LIN {X 0,Y 573.567,Z 656.189,A -85,B 0,C 180,E1 -2262.742,E2 -2262.742} C_VEL
LIN {X 0,Y 573.743,Z 644.019,A -85,B 0,C 180,E1 -2263.819,E2 -2263.819} C_VEL
LIN {X 0,Y 573.96,Z 630.902,A -85,B 0,C 180,E1 -2264.781,E2 -2264.781} C_VEL
LIN {X 0,Y 574.111,Z 618.515,A -85,B 0,C 180,E1 -2265.532,E2 -2265.532} C_VEL
LIN {X 0,Y 574.333,Z 603.831,A -85,B 0,C 180,E1 -2266.255,E2 -2266.255} C_VEL
LIN {X 0,Y 574.538,Z 589.615,A -85,B 0,C 180,E1 -2266.798,E2 -2266.798} C_VEL
LIN {X 0,Y 574.7,Z 574.63,A -85,B 0,C 180,E1 -2267.221,E2 -2267.221} C_VEL
LIN {X 0,Y 574.751,Z 559.735,A -85,B 0,C 180,E1 -2267.502,E2 -2267.502} C_VEL
LIN {X 0,Y 575.142,Z 404.764,A -85,B 0,C 180,E1 -2269.493,E2 -2269.493} C_VEL
LIN {X 0,Y 574.007,Z 398.748,A -85,B 0,C 180,E1 -2269.627,E2 -2269.627} C_VEL
LIN {X 0,Y 574.33,Z 374.816,A -85,B 0,C 180,E1 -2272.483,E2 -2272.483} C_VEL
LIN {X 0,Y 574.662,Z 351.3,A -85,B 0,C 180,E1 -2275.343,E2 -2275.343} C_VEL
LIN {X 0,Y 574.14,Z 346.557,A -85,B 0,C 180,E1 -2275.952,E2 -2275.952} C_VEL
LIN {X 0,Y 573.222,Z 342.711,A -85,B 0,C 180,E1 -2276.489,E2 -2276.489} C_VEL
LIN {X 0,Y 573.243,Z 342.7,A -85,B 0,C 180,E1 -2279.367,E2 -2279.367} C_VEL
LIN {X 0,Y 573.248,Z 342.707,A -85,B 0,C 180,E1 -2282.228,E2 -2282.228} C_VEL
LIN {X 0,Y 573.221,Z 342.706,A -85,B 0,C 180,E1 -2284.769,E2 -2284.769} C_VEL
LIN {X 0,Y 573.22,Z 342.704,A -85,B 0,C 180,E1 -2287.809,E2 -2287.809} C_VEL
LIN {X 0,Y 573.245,Z 342.706,A -85,B 0,C 180,E1 -2290.525,E2 -2290.525} C_VEL
LIN {X 0,Y 573.206,Z 342.703,A -85,B 0,C 180,E1 -2293.362,E2 -2293.362} C_VEL
LIN {X 0,Y 573.205,Z 342.713,A -85,B 0,C 180,E1 -2296.335,E2 -2296.335} C_VEL
LIN {X 0,Y 573.205,Z 342.711,A -85,B 0,C 180,E1 -2298.541,E2 -2298.541} C_VEL
LIN {X 0,Y 573.232,Z 342.7,A -85,B 0,C 180,E1 -2301.298,E2 -2301.298} C_VEL
LIN {X 0,Y 573.187,Z 342.708,A -85,B 0,C 180,E1 -2304.022,E2 -2304.022} C_VEL
LIN {X 0,Y 573.254,Z 342.705,A -85,B 0,C 180,E1 -2306.517,E2 -2306.517} C_VEL
LIN {X 0,Y 573.22,Z 342.699,A -85,B 0,C 180,E1 -2309.12,E2 -2309.12} C_VEL
LIN {X 0,Y 573.218,Z 342.705,A -85,B 0,C 180,E1 -2311.978,E2 -2311.978} C_VEL
LIN {X 0,Y 573.235,Z 342.707,A -85,B 0,C 180,E1 -2314.589,E2 -2314.589} C_VEL
LIN {X 0,Y 573.22,Z 342.701,A -85,B 0,C 180,E1 -2317.662,E2 -2317.662} C_VEL
LIN {X 0,Y 573.235,Z 342.702,A -85,B 0,C 180,E1 -2319.923,E2 -2319.923} C_VEL
LIN {X 0,Y 573.239,Z 342.702,A -85,B 0,C 180,E1 -2322.888,E2 -2322.888} C_VEL
LIN {X 0,Y 573.259,Z 342.698,A -85,B 0,C 180,E1 -2325.807,E2 -2325.807} C_VEL
LIN {X 0,Y 573.265,Z 342.701,A -85,B 0,C 180,E1 -2328.745,E2 -2328.745} C_VEL
LIN {X 0,Y 573.25,Z 342.697,A -85,B 0,C 180,E1 -2331.54,E2 -2331.54} C_VEL
LIN {X 0,Y 573.281,Z 342.703,A -85,B 0,C 180,E1 -2334.372,E2 -2334.372} C_VEL
LIN {X 0,Y 573.311,Z 342.692,A -85,B 0,C 180,E1 -2337.893,E2 -2337.893} C_VEL
LIN {X 0,Y 573.327,Z 342.694,A -85,B 0,C 180,E1 -2340.703,E2 -2340.703} C_VEL
LIN {X 0,Y 573.293,Z 342.696,A -85,B 0,C 180,E1 -2342.811,E2 -2342.811} C_VEL
LIN {X 0,Y 573.275,Z 342.695,A -85,B 0,C 180,E1 -2345.629,E2 -2345.629} C_VEL
LIN {X 0,Y 573.254,Z 342.706,A -85,B 0,C 180,E1 -2348.46,E2 -2348.46} C_VEL
LIN {X 0,Y 573.275,Z 342.694,A -85,B 0,C 180,E1 -2351.312,E2 -2351.312} C_VEL
LIN {X 0,Y 573.284,Z 342.703,A -85,B 0,C 180,E1 -2354.424,E2 -2354.424} C_VEL
LIN {X 0,Y 573.258,Z 342.698,A -85,B 0,C 180,E1 -2357.112,E2 -2357.112} C_VEL
LIN {X 0,Y 573.242,Z 342.698,A -85,B 0,C 180,E1 -2360.077,E2 -2360.077} C_VEL
LIN {X 0,Y 573.233,Z 342.707,A -85,B 0,C 180,E1 -2362.338,E2 -2362.338} C_VEL
LIN {X 0,Y 573.228,Z 342.703,A -85,B 0,C 180,E1 -2364.384,E2 -2364.384} C_VEL
LIN {X 0,Y 572.583,Z 342.786,A -85,B 0,C 180,E1 -2364.971,E2 -2364.971} C_VEL
LIN {X 0,Y 569.726,Z 343.142,A -85,B 0,C 180,E1 -2365.922,E2 -2365.922} C_VEL
LIN {X 0,Y 567.296,Z 343.446,A -85,B 0,C 180,E1 -2366.687,E2 -2366.687} C_VEL
LIN {X 0,Y 566.25,Z 343.57,A -85,B 0,C 180,E1 -2367.279,E2 -2367.279} C_VEL
LIN {X 0,Y 566.165,Z 343.58,A -85,B 0,C 180,E1 -2367.479,E2 -2367.479} C_VEL
LIN {X 0,Y 566.202,Z 343.576,A -85,B 0,C 180,E1 -2369.769,E2 -2369.769} C_VEL
LIN {X 0,Y 566.206,Z 343.582,A -85,B 0,C 180,E1 -2372.43,E2 -2372.43} C_VEL
LIN {X 0,Y 566.173,Z 343.58,A -85,B 0,C 180,E1 -2374.988,E2 -2374.988} C_VEL
LIN {X 0,Y 566.19,Z 343.578,A -85,B 0,C 180,E1 -2377.462,E2 -2377.462} C_VEL
LIN {X 0,Y 566.21,Z 343.578,A -85,B 0,C 180,E1 -2380.199,E2 -2380.199} C_VEL
LIN {X 0,Y 566.19,Z 343.58,A -85,B 0,C 180,E1 -2383.056,E2 -2383.056} C_VEL
LIN {X 0,Y 566.197,Z 343.579,A -85,B 0,C 180,E1 -2386.05,E2 -2386.05} C_VEL
LIN {X 0,Y 566.207,Z 343.577,A -85,B 0,C 180,E1 -2389.215,E2 -2389.215} C_VEL
LIN {X 0,Y 566.184,Z 343.579,A -85,B 0,C 180,E1 -2391.637,E2 -2391.637} C_VEL
LIN {X 0,Y 566.153,Z 343.589,A -85,B 0,C 180,E1 -2394.307,E2 -2394.307} C_VEL
LIN {X 0,Y 566.245,Z 343.761,A -85,B 0,C 180,E1 -2396.718,E2 -2396.718} C_VEL
LIN {X 0,Y 567.126,Z 349.166,A -85,B 0,C 180,E1 -2397.534,E2 -2397.534} C_VEL
LIN {X 0,Y 566.884,Z 367.95,A -85,B 0,C 180,E1 -2400.188,E2 -2400.188} C_VEL
LIN {X 0,Y 568.456,Z 375.277,A -85,B 0,C 180,E1 -2400.346,E2 -2400.346} C_VEL
LIN {X 0,Y 567.962,Z 533.328,A -85,B 0,C 180,E1 -2402.415,E2 -2402.415} C_VEL
LIN {X 0,Y 567.836,Z 548.985,A -85,B 0,C 180,E1 -2402.773,E2 -2402.773} C_VEL
LIN {X 0,Y 567.605,Z 564.367,A -85,B 0,C 180,E1 -2403.281,E2 -2403.281} C_VEL
LIN {X 0,Y 567.381,Z 578.806,A -85,B 0,C 180,E1 -2403.913,E2 -2403.913} C_VEL
LIN {X 0,Y 567.142,Z 592.847,A -85,B 0,C 180,E1 -2404.69,E2 -2404.69} C_VEL
LIN {X 0,Y 566.884,Z 605.684,A -85,B 0,C 180,E1 -2405.558,E2 -2405.558} C_VEL
LIN {X 0,Y 566.664,Z 618.585,A -85,B 0,C 180,E1 -2406.617,E2 -2406.617} C_VEL
LIN {X 0,Y 566.45,Z 630.204,A -85,B 0,C 180,E1 -2407.764,E2 -2407.764} C_VEL
LIN {X 0,Y 566.259,Z 639.933,A -85,B 0,C 180,E1 -2408.904,E2 -2408.904} C_VEL
LIN {X 0,Y 566.132,Z 649.359,A -85,B 0,C 180,E1 -2410.228,E2 -2410.228} C_VEL
LIN {X 0,Y 566.048,Z 657.113,A -85,B 0,C 180,E1 -2411.542,E2 -2411.542} C_VEL
LIN {X 0,Y 565.971,Z 663.975,A -85,B 0,C 180,E1 -2412.972,E2 -2412.972} C_VEL
LIN {X 0,Y 565.911,Z 669.753,A -85,B 0,C 180,E1 -2414.514,E2 -2414.514} C_VEL
LIN {X 0,Y 565.895,Z 672.935,A -85,B 0,C 180,E1 -2415.63,E2 -2415.63} C_VEL
LIN {X 0,Y 565.847,Z 676.002,A -85,B 0,C 180,E1 -2417.081,E2 -2417.081} C_VEL
LIN {X 0,Y 565.877,Z 677.854,A -85,B 0,C 180,E1 -2418.538,E2 -2418.538} C_VEL
LIN {X 0,Y 565.88,Z 678.493,A -85,B 0,C 180,E1 -2419.987,E2 -2419.987} C_VEL
LIN {X 0,Y 565.849,Z 677.938,A -85,B 0,C 180,E1 -2421.429,E2 -2421.429} C_VEL
LIN {X 0,Y 565.883,Z 676.229,A -85,B 0,C 180,E1 -2422.866,E2 -2422.866} C_VEL
LIN {X 0,Y 565.921,Z 673.341,A -85,B 0,C 180,E1 -2424.298,E2 -2424.298} C_VEL
LIN {X 0,Y 565.956,Z 669.229,A -85,B 0,C 180,E1 -2425.727,E2 -2425.727} C_VEL
LIN {X 0,Y 565.92,Z 663.819,A -85,B 0,C 180,E1 -2427.153,E2 -2427.153} C_VEL
LIN {X 0,Y 566.009,Z 656.958,A -85,B 0,C 180,E1 -2428.577,E2 -2428.577} C_VEL
LIN {X 0,Y 566.155,Z 648.451,A -85,B 0,C 180,E1 -2430,E2 -2430} C_VEL
LIN {X 0,Y 566.298,Z 639.466,A -85,B 0,C 180,E1 -2431.245,E2 -2431.245} C_VEL
LIN {X 0,Y 566.455,Z 628.688,A -85,B 0,C 180,E1 -2432.489,E2 -2432.489} C_VEL
LIN {X 0,Y 566.681,Z 617.671,A -85,B 0,C 180,E1 -2433.555,E2 -2433.555} C_VEL
LIN {X 0,Y 566.936,Z 605.649,A -85,B 0,C 180,E1 -2434.533,E2 -2434.533} C_VEL
LIN {X 0,Y 567.165,Z 592.496,A -85,B 0,C 180,E1 -2435.422,E2 -2435.422} C_VEL
LIN {X 0,Y 567.403,Z 579.639,A -85,B 0,C 180,E1 -2436.133,E2 -2436.133} C_VEL
LIN {X 0,Y 567.611,Z 565.672,A -85,B 0,C 180,E1 -2436.755,E2 -2436.755} C_VEL
LIN {X 0,Y 567.786,Z 550.58,A -85,B 0,C 180,E1 -2437.27,E2 -2437.27} C_VEL
LIN {X 0,Y 567.906,Z 535.508,A -85,B 0,C 180,E1 -2437.632,E2 -2437.632} C_VEL
LIN {X 0,Y 568.033,Z 511.55,A -85,B 0,C 180,E1 -2437.976,E2 -2437.976} C_VEL
LIN {X 0,Y 568.479,Z 375.352,A -85,B 0,C 180,E1 -2439.742,E2 -2439.742} C_VEL
LIN {X 0,Y 566.9,Z 367.922,A -85,B 0,C 180,E1 -2439.905,E2 -2439.905} C_VEL
LIN {X 0,Y 567.179,Z 349.374,A -85,B 0,C 180,E1 -2442.524,E2 -2442.524} C_VEL
LIN {X 0,Y 566.178,Z 343.589,A -85,B 0,C 180,E1 -2443.413,E2 -2443.413} C_VEL
LIN {X 0,Y 566.185,Z 343.585,A -85,B 0,C 180,E1 -2445.848,E2 -2445.848} C_VEL
LIN {X 0,Y 566.18,Z 343.582,A -85,B 0,C 180,E1 -2448.079,E2 -2448.079} C_VEL
LIN {X 0,Y 566.206,Z 343.575,A -85,B 0,C 180,E1 -2450.338,E2 -2450.338} C_VEL
LIN {X 0,Y 566.171,Z 343.586,A -85,B 0,C 180,E1 -2453.28,E2 -2453.28} C_VEL
LIN {X 0,Y 566.198,Z 343.583,A -85,B 0,C 180,E1 -2455.75,E2 -2455.75} C_VEL
LIN {X 0,Y 566.163,Z 343.582,A -85,B 0,C 180,E1 -2458.193,E2 -2458.193} C_VEL
LIN {X 0,Y 566.189,Z 343.58,A -85,B 0,C 180,E1 -2461.075,E2 -2461.075} C_VEL
LIN {X 0,Y 566.216,Z 343.581,A -85,B 0,C 180,E1 -2463.734,E2 -2463.734} C_VEL
LIN {X 0,Y 566.151,Z 343.581,A -85,B 0,C 180,E1 -2466.574,E2 -2466.574} C_VEL
LIN {X 0,Y 566.212,Z 343.58,A -85,B 0,C 180,E1 -2469.274,E2 -2469.274} C_VEL
LIN {X 0,Y 566.173,Z 343.581,A -85,B 0,C 180,E1 -2472.091,E2 -2472.091} C_VEL
LIN {X 0,Y 566.168,Z 343.582,A -85,B 0,C 180,E1 -2475.037,E2 -2475.037} C_VEL
LIN {X 0,Y 566.183,Z 343.582,A -85,B 0,C 180,E1 -2477.909,E2 -2477.909} C_VEL
LIN {X 0,Y 566.211,Z 343.574,A -85,B 0,C 180,E1 -2480.725,E2 -2480.725} C_VEL
LIN {X 0,Y 566.178,Z 343.586,A -85,B 0,C 180,E1 -2483.428,E2 -2483.428} C_VEL
LIN {X 0,Y 566.201,Z 343.576,A -85,B 0,C 180,E1 -2486.268,E2 -2486.268} C_VEL
LIN {X 0,Y 566.189,Z 343.579,A -85,B 0,C 180,E1 -2488.924,E2 -2488.924} C_VEL
LIN {X 0,Y 566.191,Z 343.578,A -85,B 0,C 180,E1 -2491.856,E2 -2491.856} C_VEL
LIN {X 0,Y 566.188,Z 343.572,A -85,B 0,C 180,E1 -2494.249,E2 -2494.249} C_VEL
LIN {X 0,Y 566.17,Z 343.578,A -85,B 0,C 180,E1 -2496.72,E2 -2496.72} C_VEL
LIN {X 0,Y 566.207,Z 343.584,A -85,B 0,C 180,E1 -2499.662,E2 -2499.662} C_VEL
LIN {X 0,Y 566.183,Z 343.58,A -85,B 0,C 180,E1 -2501.921,E2 -2501.921} C_VEL
LIN {X 0,Y 566.19,Z 343.579,A -85,B 0,C 180,E1 -2504.152,E2 -2504.152} C_VEL
LIN {X 0,Y 566.185,Z 343.578,A -85,B 0,C 180,E1 -2506.358,E2 -2506.358} C_VEL
LIN {X 0,Y 566.236,Z 343.574,A -85,B 0,C 180,E1 -2509.27,E2 -2509.27} C_VEL
LIN {X 0,Y 566.194,Z 343.578,A -85,B 0,C 180,E1 -2512.152,E2 -2512.152} C_VEL
LIN {X 0,Y 566.265,Z 343.567,A -85,B 0,C 180,E1 -2515.016,E2 -2515.016} C_VEL
LIN {X 0,Y 566.282,Z 343.571,A -85,B 0,C 180,E1 -2517.866,E2 -2517.866} C_VEL
LIN {X 0,Y 566.29,Z 343.567,A -85,B 0,C 180,E1 -2520,E2 -2520} C_VEL
LIN {X 0,Y 566.255,Z 343.568,A -85,B 0,C 180,E1 -2522.845,E2 -2522.845} C_VEL
LIN {X 0,Y 566.248,Z 343.578,A -85,B 0,C 180,E1 -2525.698,E2 -2525.698} C_VEL
LIN {X 0,Y 566.2,Z 343.575,A -85,B 0,C 180,E1 -2528.566,E2 -2528.566} C_VEL
LIN {X 0,Y 566.242,Z 343.578,A -85,B 0,C 180,E1 -2531.454,E2 -2531.454} C_VEL
LIN {X 0,Y 566.227,Z 343.572,A -85,B 0,C 180,E1 -2534.502,E2 -2534.502} C_VEL
LIN {X 0,Y 566.162,Z 343.585,A -85,B 0,C 180,E1 -2537.333,E2 -2537.333} C_VEL
LIN {X 0,Y 566.201,Z 343.584,A -85,B 0,C 180,E1 -2539.581,E2 -2539.581} C_VEL
LIN {X 0,Y 566.186,Z 343.582,A -85,B 0,C 180,E1 -2541.863,E2 -2541.863} C_VEL
LIN {X 0,Y 566.183,Z 343.579,A -85,B 0,C 180,E1 -2545.022,E2 -2545.022} C_VEL
LIN {X 0,Y 566.168,Z 343.584,A -85,B 0,C 180,E1 -2547.341,E2 -2547.341} C_VEL
LIN {X 0,Y 566.172,Z 343.587,A -85,B 0,C 180,E1 -2549.77,E2 -2549.77} C_VEL
LIN {X 0,Y 566.2,Z 343.576,A -85,B 0,C 180,E1 -2552.429,E2 -2552.429} C_VEL
LIN {X 0,Y 566.169,Z 343.581,A -85,B 0,C 180,E1 -2554.987,E2 -2554.987} C_VEL
LIN {X 0,Y 566.186,Z 343.585,A -85,B 0,C 180,E1 -2557.461,E2 -2557.461} C_VEL
LIN {X 0,Y 566.206,Z 343.577,A -85,B 0,C 180,E1 -2560.199,E2 -2560.199} C_VEL
LIN {X 0,Y 566.177,Z 343.58,A -85,B 0,C 180,E1 -2563.056,E2 -2563.056} C_VEL
LIN {X 0,Y 566.158,Z 343.585,A -85,B 0,C 180,E1 -2566.053,E2 -2566.053} C_VEL
LIN {X 0,Y 566.158,Z 343.582,A -85,B 0,C 180,E1 -2568.859,E2 -2568.859} C_VEL
LIN {X 0,Y 566.202,Z 343.584,A -85,B 0,C 180,E1 -2571.443,E2 -2571.443} C_VEL
LIN {X 0,Y 566.14,Z 343.585,A -85,B 0,C 180,E1 -2574.306,E2 -2574.306} C_VEL
LIN {X 0,Y 566.203,Z 343.577,A -85,B 0,C 180,E1 -2576.897,E2 -2576.897} C_VEL
LIN {X 0,Y 566.175,Z 343.586,A -85,B 0,C 180,E1 -2579.407,E2 -2579.407} C_VEL
LIN {X 0,Y 566.187,Z 343.587,A -85,B 0,C 180,E1 -2581.856,E2 -2581.856} C_VEL
LIN {X 0,Y 566.174,Z 343.693,A -85,B 0,C 180,E1 -2583.323,E2 -2583.323} C_VEL
LIN {X 0,Y 567.812,Z 351.159,A -85,B 0,C 180,E1 -2584.329,E2 -2584.329} C_VEL
LIN {X 0,Y 567.553,Z 371.68,A -85,B 0,C 180,E1 -2586.849,E2 -2586.849} C_VEL
LIN {X 0,Y 567.151,Z 396.606,A -85,B 0,C 180,E1 -2589.868,E2 -2589.868} C_VEL
LIN {X 0,Y 567.116,Z 398.903,A -85,B 0,C 180,E1 -2590.142,E2 -2590.142} C_VEL
LIN {X 0,Y 568.488,Z 406.26,A -85,B 0,C 180,E1 -2590.289,E2 -2590.289} C_VEL
LIN {X 0,Y 567.984,Z 564.94,A -85,B 0,C 180,E1 -2592.364,E2 -2592.364} C_VEL
LIN {X 0,Y 567.834,Z 580.701,A -85,B 0,C 180,E1 -2592.72,E2 -2592.72} C_VEL
LIN {X 0,Y 567.627,Z 596.036,A -85,B 0,C 180,E1 -2593.223,E2 -2593.223} C_VEL
LIN {X 0,Y 567.461,Z 609.77,A -85,B 0,C 180,E1 -2593.82,E2 -2593.82} C_VEL
LIN {X 0,Y 567.151,Z 623.244,A -85,B 0,C 180,E1 -2594.548,E2 -2594.548} C_VEL
LIN {X 0,Y 566.932,Z 635.518,A -85,B 0,C 180,E1 -2595.359,E2 -2595.359} C_VEL
LIN {X 0,Y 566.672,Z 648.29,A -85,B 0,C 180,E1 -2596.37,E2 -2596.37} C_VEL
LIN {X 0,Y 566.491,Z 659.748,A -85,B 0,C 180,E1 -2597.461,E2 -2597.461} C_VEL
LIN {X 0,Y 566.268,Z 670.311,A -85,B 0,C 180,E1 -2598.659,E2 -2598.659} C_VEL
LIN {X 0,Y 566.209,Z 678.856,A -85,B 0,C 180,E1 -2599.812,E2 -2599.812} C_VEL
LIN {X 0,Y 566.057,Z 686.734,A -85,B 0,C 180,E1 -2601.072,E2 -2601.072} C_VEL
LIN {X 0,Y 565.997,Z 694.089,A -85,B 0,C 180,E1 -2602.508,E2 -2602.508} C_VEL
LIN {X 0,Y 565.958,Z 699.923,A -85,B 0,C 180,E1 -2603.941,E2 -2603.941} C_VEL
LIN {X 0,Y 565.866,Z 703.385,A -85,B 0,C 180,E1 -2605.012,E2 -2605.012} C_VEL
LIN {X 0,Y 565.91,Z 706.89,A -85,B 0,C 180,E1 -2606.44,E2 -2606.44} C_VEL
LIN {X 0,Y 565.839,Z 709.192,A -85,B 0,C 180,E1 -2607.865,E2 -2607.865} C_VEL
LIN {X 0,Y 565.836,Z 710.349,A -85,B 0,C 180,E1 -2609.288,E2 -2609.288} C_VEL
LIN {X 0,Y 565.836,Z 710.349,A -85,B 0,C 180,E1 -2610.712,E2 -2610.712} C_VEL
LIN {X 0,Y 565.838,Z 709.19,A -85,B 0,C 180,E1 -2612.135,E2 -2612.135} C_VEL
LIN {X 0,Y 565.91,Z 706.887,A -85,B 0,C 180,E1 -2613.56,E2 -2613.56} C_VEL
LIN {X 0,Y 565.866,Z 703.386,A -85,B 0,C 180,E1 -2614.988,E2 -2614.988} C_VEL
LIN {X 0,Y 565.942,Z 698.609,A -85,B 0,C 180,E1 -2616.417,E2 -2616.417} C_VEL
LIN {X 0,Y 566.014,Z 692.422,A -85,B 0,C 180,E1 -2617.85,E2 -2617.85} C_VEL
LIN {X 0,Y 566.071,Z 684.647,A -85,B 0,C 180,E1 -2619.288,E2 -2619.288} C_VEL
LIN {X 0,Y 566.239,Z 676.369,A -85,B 0,C 180,E1 -2620.549,E2 -2620.549} C_VEL
LIN {X 0,Y 566.367,Z 666.391,A -85,B 0,C 180,E1 -2621.815,E2 -2621.815} C_VEL
LIN {X 0,Y 566.585,Z 656.188,A -85,B 0,C 180,E1 -2622.901,E2 -2622.901} C_VEL
LIN {X 0,Y 566.8,Z 644.019,A -85,B 0,C 180,E1 -2623.992,E2 -2623.992} C_VEL
LIN {X 0,Y 567.037,Z 631.339,A -85,B 0,C 180,E1 -2624.936,E2 -2624.936} C_VEL
LIN {X 0,Y 567.23,Z 618.513,A -85,B 0,C 180,E1 -2625.726,E2 -2625.726} C_VEL
LIN {X 0,Y 567.515,Z 603.829,A -85,B 0,C 180,E1 -2626.456,E2 -2626.456} C_VEL
LIN {X 0,Y 567.726,Z 589.614,A -85,B 0,C 180,E1 -2627.005,E2 -2627.005} C_VEL
LIN {X 0,Y 567.922,Z 575.27,A -85,B 0,C 180,E1 -2627.417,E2 -2627.417} C_VEL
LIN {X 0,Y 567.983,Z 560.821,A -85,B 0,C 180,E1 -2627.7,E2 -2627.7} C_VEL
LIN {X 0,Y 568.462,Z 405.814,A -85,B 0,C 180,E1 -2629.718,E2 -2629.718} C_VEL
LIN {X 0,Y 567.135,Z 398.804,A -85,B 0,C 180,E1 -2629.868,E2 -2629.868} C_VEL
LIN {X 0,Y 567.494,Z 374.816,A -85,B 0,C 180,E1 -2632.769,E2 -2632.769} C_VEL
LIN {X 0,Y 567.834,Z 352.86,A -85,B 0,C 180,E1 -2635.457,E2 -2635.457} C_VEL
LIN {X 0,Y 567.193,Z 347.931,A -85,B 0,C 180,E1 -2636.096,E2 -2636.096} C_VEL
LIN {X 0,Y 566.168,Z 343.589,A -85,B 0,C 180,E1 -2636.718,E2 -2636.718} C_VEL
LIN {X 0,Y 566.193,Z 343.579,A -85,B 0,C 180,E1 -2639.67,E2 -2639.67} C_VEL
LIN {X 0,Y 566.201,Z 343.586,A -85,B 0,C 180,E1 -2642.43,E2 -2642.43} C_VEL
LIN {X 0,Y 566.165,Z 343.583,A -85,B 0,C 180,E1 -2644.987,E2 -2644.987} C_VEL
LIN {X 0,Y 566.185,Z 343.578,A -85,B 0,C 180,E1 -2647.462,E2 -2647.462} C_VEL
LIN {X 0,Y 566.205,Z 343.582,A -85,B 0,C 180,E1 -2650.199,E2 -2650.199} C_VEL
LIN {X 0,Y 566.186,Z 343.579,A -85,B 0,C 180,E1 -2653.056,E2 -2653.056} C_VEL
LIN {X 0,Y 566.156,Z 343.587,A -85,B 0,C 180,E1 -2656.053,E2 -2656.053} C_VEL
LIN {X 0,Y 566.157,Z 343.585,A -85,B 0,C 180,E1 -2658.859,E2 -2658.859} C_VEL
LIN {X 0,Y 566.202,Z 343.576,A -85,B 0,C 180,E1 -2661.443,E2 -2661.443} C_VEL
LIN {X 0,Y 566.142,Z 343.588,A -85,B 0,C 180,E1 -2664.307,E2 -2664.307} C_VEL
LIN {X 0,Y 566.211,Z 343.577,A -85,B 0,C 180,E1 -2666.897,E2 -2666.897} C_VEL
LIN {X 0,Y 566.169,Z 343.575,A -85,B 0,C 180,E1 -2669.407,E2 -2669.407} C_VEL
LIN {X 0,Y 566.188,Z 343.579,A -85,B 0,C 180,E1 -2671.856,E2 -2671.856} C_VEL
LIN {X 0,Y 566.195,Z 343.583,A -85,B 0,C 180,E1 -2674.25,E2 -2674.25} C_VEL
LIN {X 0,Y 566.166,Z 343.585,A -85,B 0,C 180,E1 -2676.72,E2 -2676.72} C_VEL
LIN {X 0,Y 566.202,Z 343.576,A -85,B 0,C 180,E1 -2679.663,E2 -2679.663} C_VEL
LIN {X 0,Y 566.177,Z 343.581,A -85,B 0,C 180,E1 -2681.921,E2 -2681.921} C_VEL
LIN {X 0,Y 566.188,Z 343.58,A -85,B 0,C 180,E1 -2684.89,E2 -2684.89} C_VEL
LIN {X 0,Y 566.213,Z 343.575,A -85,B 0,C 180,E1 -2687.819,E2 -2687.819} C_VEL
LIN {X 0,Y 566.174,Z 343.582,A -85,B 0,C 180,E1 -2689.992,E2 -2689.992} C_VEL
LIN {X 0,Y 566.212,Z 343.578,A -85,B 0,C 180,E1 -2692.87,E2 -2692.87} C_VEL
LIN {X 0,Y 566.262,Z 343.569,A -85,B 0,C 180,E1 -2695.016,E2 -2695.016} C_VEL
LIN {X 0,Y 566.281,Z 343.568,A -85,B 0,C 180,E1 -2697.867,E2 -2697.867} C_VEL
LIN {X 0,Y 566.297,Z 343.57,A -85,B 0,C 180,E1 -2700.711,E2 -2700.711} C_VEL
LIN {X 0,Y 566.259,Z 343.571,A -85,B 0,C 180,E1 -2702.846,E2 -2702.846} C_VEL
LIN {X 0,Y 566.245,Z 343.571,A -85,B 0,C 180,E1 -2705.699,E2 -2705.699} C_VEL
LIN {X 0,Y 566.204,Z 343.584,A -85,B 0,C 180,E1 -2708.566,E2 -2708.566} C_VEL
LIN {X 0,Y 566.245,Z 343.569,A -85,B 0,C 180,E1 -2711.455,E2 -2711.455} C_VEL
LIN {X 0,Y 566.237,Z 343.58,A -85,B 0,C 180,E1 -2714.506,E2 -2714.506} C_VEL
LIN {X 0,Y 566.196,Z 343.576,A -85,B 0,C 180,E1 -2717.332,E2 -2717.332} C_VEL
LIN {X 0,Y 566.209,Z 343.578,A -85,B 0,C 180,E1 -2720.338,E2 -2720.338} C_VEL
LIN {X 0,Y 566.171,Z 343.58,A -85,B 0,C 180,E1 -2723.281,E2 -2723.281} C_VEL
LIN {X 0,Y 566.192,Z 343.574,A -85,B 0,C 180,E1 -2725.751,E2 -2725.751} C_VEL
LIN {X 0,Y 566.165,Z 343.58,A -85,B 0,C 180,E1 -2727.479,E2 -2727.479} C_VEL
LIN {X 0,Y 565.498,Z 343.668,A -85,B 0,C 180,E1 -2728.073,E2 -2728.073} C_VEL
LIN {X 0,Y 562.649,Z 344.021,A -85,B 0,C 180,E1 -2729.037,E2 -2729.037} C_VEL
LIN {X 0,Y 560.246,Z 344.32,A -85,B 0,C 180,E1 -2729.813,E2 -2729.813} C_VEL
LIN {X 0,Y 559.221,Z 344.452,A -85,B 0,C 180,E1 -2730.412,E2 -2730.412} C_VEL
LIN {X 0,Y 559.14,Z 344.456,A -85,B 0,C 180,E1 -2730.615,E2 -2730.615} C_VEL
LIN {X 0,Y 559.156,Z 344.461,A -85,B 0,C 180,E1 -2732.716,E2 -2732.716} C_VEL
LIN {X 0,Y 559.121,Z 344.455,A -85,B 0,C 180,E1 -2735.325,E2 -2735.325} C_VEL
LIN {X 0,Y 559.129,Z 344.46,A -85,B 0,C 180,E1 -2738.018,E2 -2738.018} C_VEL
LIN {X 0,Y 559.131,Z 344.462,A -85,B 0,C 180,E1 -2740.815,E2 -2740.815} C_VEL
LIN {X 0,Y 559.134,Z 344.458,A -85,B 0,C 180,E1 -2743.195,E2 -2743.195} C_VEL
LIN {X 0,Y 559.139,Z 344.461,A -85,B 0,C 180,E1 -2746.266,E2 -2746.266} C_VEL
LIN {X 0,Y 559.159,Z 344.456,A -85,B 0,C 180,E1 -2749.188,E2 -2749.188} C_VEL
LIN {X 0,Y 559.132,Z 344.46,A -85,B 0,C 180,E1 -2751.982,E2 -2751.982} C_VEL
LIN {X 0,Y 559.131,Z 344.466,A -85,B 0,C 180,E1 -2754.788,E2 -2754.788} C_VEL
LIN {X 0,Y 559.206,Z 344.622,A -85,B 0,C 180,E1 -2756.507,E2 -2756.507} C_VEL
LIN {X 0,Y 560.22,Z 350.036,A -85,B 0,C 180,E1 -2757.355,E2 -2757.355} C_VEL
LIN {X 0,Y 559.978,Z 367.88,A -85,B 0,C 180,E1 -2759.923,E2 -2759.923} C_VEL
LIN {X 0,Y 561.822,Z 377.426,A -85,B 0,C 180,E1 -2760.132,E2 -2760.132} C_VEL
LIN {X 0,Y 561.206,Z 533.216,A -85,B 0,C 180,E1 -2762.194,E2 -2762.194} C_VEL
LIN {X 0,Y 561.059,Z 548.754,A -85,B 0,C 180,E1 -2762.551,E2 -2762.551} C_VEL
LIN {X 0,Y 560.78,Z 563.702,A -85,B 0,C 180,E1 -2763.044,E2 -2763.044} C_VEL
LIN {X 0,Y 560.539,Z 578.009,A -85,B 0,C 180,E1 -2763.671,E2 -2763.671} C_VEL
LIN {X 0,Y 560.252,Z 591.626,A -85,B 0,C 180,E1 -2764.421,E2 -2764.421} C_VEL
LIN {X 0,Y 559.979,Z 605.146,A -85,B 0,C 180,E1 -2765.336,E2 -2765.336} C_VEL
LIN {X 0,Y 559.741,Z 617.059,A -85,B 0,C 180,E1 -2766.31,E2 -2766.31} C_VEL
LIN {X 0,Y 559.452,Z 628.959,A -85,B 0,C 180,E1 -2767.471,E2 -2767.471} C_VEL
LIN {X 0,Y 559.219,Z 638.852,A -85,B 0,C 180,E1 -2768.626,E2 -2768.626} C_VEL
LIN {X 0,Y 559.104,Z 648.484,A -85,B 0,C 180,E1 -2769.969,E2 -2769.969} C_VEL
LIN {X 0,Y 558.975,Z 656.374,A -85,B 0,C 180,E1 -2771.3,E2 -2771.3} C_VEL
LIN {X 0,Y 558.913,Z 661.986,A -85,B 0,C 180,E1 -2772.435,E2 -2772.435} C_VEL
LIN {X 0,Y 558.834,Z 668.026,A -85,B 0,C 180,E1 -2773.938,E2 -2773.938} C_VEL
LIN {X 0,Y 558.806,Z 672.584,A -85,B 0,C 180,E1 -2775.432,E2 -2775.432} C_VEL
LIN {X 0,Y 558.749,Z 675.799,A -85,B 0,C 180,E1 -2776.914,E2 -2776.914} C_VEL
LIN {X 0,Y 558.777,Z 677.745,A -85,B 0,C 180,E1 -2778.391,E2 -2778.391} C_VEL
LIN {X 0,Y 558.777,Z 678.466,A -85,B 0,C 180,E1 -2779.858,E2 -2779.858} C_VEL
LIN {X 0,Y 558.763,Z 678.022,A -85,B 0,C 180,E1 -2781.319,E2 -2781.319} C_VEL
LIN {X 0,Y 558.794,Z 676.425,A -85,B 0,C 180,E1 -2782.775,E2 -2782.775} C_VEL
LIN {X 0,Y 558.829,Z 673.652,A -85,B 0,C 180,E1 -2784.226,E2 -2784.226} C_VEL
LIN {X 0,Y 558.861,Z 669.662,A -85,B 0,C 180,E1 -2785.673,E2 -2785.673} C_VEL
LIN {X 0,Y 558.841,Z 664.36,A -85,B 0,C 180,E1 -2787.117,E2 -2787.117} C_VEL
LIN {X 0,Y 558.927,Z 657.62,A -85,B 0,C 180,E1 -2788.559,E2 -2788.559} C_VEL
LIN {X 0,Y 559.106,Z 649.281,A -85,B 0,C 180,E1 -2790,E2 -2790} C_VEL
LIN {X 0,Y 559.254,Z 640.43,A -85,B 0,C 180,E1 -2791.26,E2 -2791.26} C_VEL
LIN {X 0,Y 559.437,Z 629.869,A -85,B 0,C 180,E1 -2792.52,E2 -2792.52} C_VEL
LIN {X 0,Y 559.69,Z 619.043,A -85,B 0,C 180,E1 -2793.6,E2 -2793.6} C_VEL
LIN {X 0,Y 559.962,Z 607.271,A -85,B 0,C 180,E1 -2794.589,E2 -2794.589} C_VEL
LIN {X 0,Y 560.263,Z 594.444,A -85,B 0,C 180,E1 -2795.489,E2 -2795.489} C_VEL
LIN {X 0,Y 560.471,Z 582.059,A -85,B 0,C 180,E1 -2796.209,E2 -2796.209} C_VEL
LIN {X 0,Y 560.743,Z 567.656,A -85,B 0,C 180,E1 -2796.884,E2 -2796.884} C_VEL
LIN {X 0,Y 560.979,Z 552.45,A -85,B 0,C 180,E1 -2797.428,E2 -2797.428} C_VEL
LIN {X 0,Y 561.135,Z 536.82,A -85,B 0,C 180,E1 -2797.824,E2 -2797.824} C_VEL
LIN {X 0,Y 561.289,Z 516.229,A -85,B 0,C 180,E1 -2798.137,E2 -2798.137} C_VEL
LIN {X 0,Y 561.705,Z 376.067,A -85,B 0,C 180,E1 -2799.98,E2 -2799.98} C_VEL
LIN {X 0,Y 560.012,Z 367.885,A -85,B 0,C 180,E1 -2800.165,E2 -2800.165} C_VEL
LIN {X 0,Y 560.244,Z 350.387,A -85,B 0,C 180,E1 -2802.681,E2 -2802.681} C_VEL
LIN {X 0,Y 559.165,Z 344.463,A -85,B 0,C 180,E1 -2803.631,E2 -2803.631} C_VEL
LIN {X 0,Y 559.143,Z 344.46,A -85,B 0,C 180,E1 -2806.053,E2 -2806.053} C_VEL
LIN {X 0,Y 559.162,Z 344.458,A -85,B 0,C 180,E1 -2809.074,E2 -2809.074} C_VEL
LIN {X 0,Y 559.159,Z 344.462,A -85,B 0,C 180,E1 -2811.549,E2 -2811.549} C_VEL
LIN {X 0,Y 559.129,Z 344.457,A -85,B 0,C 180,E1 -2814.507,E2 -2814.507} C_VEL
LIN {X 0,Y 559.137,Z 344.457,A -85,B 0,C 180,E1 -2816.904,E2 -2816.904} C_VEL
LIN {X 0,Y 559.126,Z 344.462,A -85,B 0,C 180,E1 -2819.852,E2 -2819.852} C_VEL
LIN {X 0,Y 559.158,Z 344.452,A -85,B 0,C 180,E1 -2822.715,E2 -2822.715} C_VEL
LIN {X 0,Y 559.122,Z 344.464,A -85,B 0,C 180,E1 -2825.325,E2 -2825.325} C_VEL
LIN {X 0,Y 559.129,Z 344.46,A -85,B 0,C 180,E1 -2828.018,E2 -2828.018} C_VEL
LIN {X 0,Y 559.162,Z 344.454,A -85,B 0,C 180,E1 -2829.941,E2 -2829.941} C_VEL
LIN {X 0,Y 559.144,Z 344.455,A -85,B 0,C 180,E1 -2832.745,E2 -2832.745} C_VEL
LIN {X 0,Y 559.127,Z 344.461,A -85,B 0,C 180,E1 -2835.764,E2 -2835.764} C_VEL
LIN {X 0,Y 559.129,Z 344.458,A -85,B 0,C 180,E1 -2838.226,E2 -2838.226} C_VEL
LIN {X 0,Y 559.173,Z 344.455,A -85,B 0,C 180,E1 -2841.192,E2 -2841.192} C_VEL
LIN {X 0,Y 559.12,Z 344.464,A -85,B 0,C 180,E1 -2843.787,E2 -2843.787} C_VEL
LIN {X 0,Y 559.152,Z 344.453,A -85,B 0,C 180,E1 -2846.424,E2 -2846.424} C_VEL
LIN {X 0,Y 559.154,Z 344.456,A -85,B 0,C 180,E1 -2848.98,E2 -2848.98} C_VEL
LIN {X 0,Y 559.137,Z 344.46,A -85,B 0,C 180,E1 -2851.625,E2 -2851.625} C_VEL
LIN {X 0,Y 559.142,Z 344.449,A -85,B 0,C 180,E1 -2854.822,E2 -2854.822} C_VEL
LIN {X 0,Y 559.142,Z 344.461,A -85,B 0,C 180,E1 -2857.847,E2 -2857.847} C_VEL
LIN {X 0,Y 559.196,Z 344.448,A -85,B 0,C 180,E1 -2860.494,E2 -2860.494} C_VEL
LIN {X 0,Y 559.17,Z 344.453,A -85,B 0,C 180,E1 -2863.197,E2 -2863.197} C_VEL
LIN {X 0,Y 559.161,Z 344.454,A -85,B 0,C 180,E1 -2866.183,E2 -2866.183} C_VEL
LIN {X 0,Y 559.194,Z 344.448,A -85,B 0,C 180,E1 -2869.133,E2 -2869.133} C_VEL
LIN {X 0,Y 559.147,Z 344.457,A -85,B 0,C 180,E1 -2872.052,E2 -2872.052} C_VEL
LIN {X 0,Y 559.24,Z 344.442,A -85,B 0,C 180,E1 -2874.953,E2 -2874.953} C_VEL
LIN {X 0,Y 559.253,Z 344.447,A -85,B 0,C 180,E1 -2877.839,E2 -2877.839} C_VEL
LIN {X 0,Y 559.259,Z 344.443,A -85,B 0,C 180,E1 -2880,E2 -2880} C_VEL
LIN {X 0,Y 559.223,Z 344.444,A -85,B 0,C 180,E1 -2882.881,E2 -2882.881} C_VEL
LIN {X 0,Y 559.217,Z 344.452,A -85,B 0,C 180,E1 -2885.77,E2 -2885.77} C_VEL
LIN {X 0,Y 559.164,Z 344.451,A -85,B 0,C 180,E1 -2888.674,E2 -2888.674} C_VEL
LIN {X 0,Y 559.203,Z 344.456,A -85,B 0,C 180,E1 -2891.6,E2 -2891.6} C_VEL
LIN {X 0,Y 559.183,Z 344.449,A -85,B 0,C 180,E1 -2894.587,E2 -2894.587} C_VEL
LIN {X 0,Y 559.117,Z 344.466,A -85,B 0,C 180,E1 -2897.558,E2 -2897.558} C_VEL
LIN {X 0,Y 559.164,Z 344.458,A -85,B 0,C 180,E1 -2899.837,E2 -2899.837} C_VEL
LIN {X 0,Y 559.132,Z 344.457,A -85,B 0,C 180,E1 -2902.153,E2 -2902.153} C_VEL
LIN {X 0,Y 559.142,Z 344.458,A -85,B 0,C 180,E1 -2905.178,E2 -2905.178} C_VEL
LIN {X 0,Y 559.118,Z 344.467,A -85,B 0,C 180,E1 -2907.715,E2 -2907.715} C_VEL
LIN {X 0,Y 559.137,Z 344.458,A -85,B 0,C 180,E1 -2910.183,E2 -2910.183} C_VEL
LIN {X 0,Y 559.154,Z 344.453,A -85,B 0,C 180,E1 -2912.715,E2 -2912.715} C_VEL
LIN {X 0,Y 559.118,Z 344.463,A -85,B 0,C 180,E1 -2915.325,E2 -2915.325} C_VEL
LIN {X 0,Y 559.124,Z 344.46,A -85,B 0,C 180,E1 -2918.018,E2 -2918.018} C_VEL
LIN {X 0,Y 559.159,Z 344.458,A -85,B 0,C 180,E1 -2919.941,E2 -2919.941} C_VEL
LIN {X 0,Y 559.139,Z 344.455,A -85,B 0,C 180,E1 -2922.745,E2 -2922.745} C_VEL
LIN {X 0,Y 559.124,Z 344.466,A -85,B 0,C 180,E1 -2925.764,E2 -2925.764} C_VEL
LIN {X 0,Y 559.126,Z 344.46,A -85,B 0,C 180,E1 -2928.226,E2 -2928.226} C_VEL
LIN {X 0,Y 559.169,Z 344.456,A -85,B 0,C 180,E1 -2931.192,E2 -2931.192} C_VEL
LIN {X 0,Y 559.115,Z 344.467,A -85,B 0,C 180,E1 -2933.787,E2 -2933.787} C_VEL
LIN {X 0,Y 559.147,Z 344.456,A -85,B 0,C 180,E1 -2936.424,E2 -2936.424} C_VEL
LIN {X 0,Y 559.152,Z 344.456,A -85,B 0,C 180,E1 -2938.98,E2 -2938.98} C_VEL
LIN {X 0,Y 559.133,Z 344.466,A -85,B 0,C 180,E1 -2941.625,E2 -2941.625} C_VEL
LIN {X 0,Y 559.144,Z 344.576,A -85,B 0,C 180,E1 -2943.096,E2 -2943.096} C_VEL
LIN {X 0,Y 560.986,Z 353.201,A -85,B 0,C 180,E1 -2944.272,E2 -2944.272} C_VEL
LIN {X 0,Y 560.69,Z 373.186,A -85,B 0,C 180,E1 -2946.744,E2 -2946.744} C_VEL
LIN {X 0,Y 560.26,Z 397.26,A -85,B 0,C 180,E1 -2949.689,E2 -2949.689} C_VEL
LIN {X 0,Y 560.268,Z 399.043,A -85,B 0,C 180,E1 -2949.891,E2 -2949.891} C_VEL
LIN {X 0,Y 561.819,Z 407.764,A -85,B 0,C 180,E1 -2950.065,E2 -2950.065} C_VEL
LIN {X 0,Y 561.232,Z 565.013,A -85,B 0,C 180,E1 -2952.146,E2 -2952.146} C_VEL
LIN {X 0,Y 561.073,Z 580.224,A -85,B 0,C 180,E1 -2952.492,E2 -2952.492} C_VEL
LIN {X 0,Y 560.832,Z 594.795,A -85,B 0,C 180,E1 -2952.967,E2 -2952.967} C_VEL
LIN {X 0,Y 560.659,Z 607.801,A -85,B 0,C 180,E1 -2953.524,E2 -2953.524} C_VEL
LIN {X 0,Y 560.317,Z 621.676,A -85,B 0,C 180,E1 -2954.262,E2 -2954.262} C_VEL
LIN {X 0,Y 560.021,Z 635.519,A -85,B 0,C 180,E1 -2955.174,E2 -2955.174} C_VEL
LIN {X 0,Y 559.722,Z 648.291,A -85,B 0,C 180,E1 -2956.198,E2 -2956.198} C_VEL
LIN {X 0,Y 559.516,Z 659.748,A -85,B 0,C 180,E1 -2957.302,E2 -2957.302} C_VEL
LIN {X 0,Y 559.304,Z 669.389,A -85,B 0,C 180,E1 -2958.402,E2 -2958.402} C_VEL
LIN {X 0,Y 559.168,Z 678.855,A -85,B 0,C 180,E1 -2959.682,E2 -2959.682} C_VEL
LIN {X 0,Y 559.002,Z 686.734,A -85,B 0,C 180,E1 -2960.958,E2 -2960.958} C_VEL
LIN {X 0,Y 558.92,Z 694.089,A -85,B 0,C 180,E1 -2962.413,E2 -2962.413} C_VEL
LIN {X 0,Y 558.859,Z 699.922,A -85,B 0,C 180,E1 -2963.864,E2 -2963.864} C_VEL
LIN {X 0,Y 558.787,Z 703.386,A -85,B 0,C 180,E1 -2964.949,E2 -2964.949} C_VEL
LIN {X 0,Y 558.819,Z 706.889,A -85,B 0,C 180,E1 -2966.395,E2 -2966.395} C_VEL
LIN {X 0,Y 558.744,Z 709.191,A -85,B 0,C 180,E1 -2967.837,E2 -2967.837} C_VEL
LIN {X 0,Y 558.737,Z 710.349,A -85,B 0,C 180,E1 -2969.279,E2 -2969.279} C_VEL
LIN {X 0,Y 558.737,Z 710.348,A -85,B 0,C 180,E1 -2970.721,E2 -2970.721} C_VEL
LIN {X 0,Y 558.744,Z 709.189,A -85,B 0,C 180,E1 -2972.163,E2 -2972.163} C_VEL
LIN {X 0,Y 558.819,Z 706.886,A -85,B 0,C 180,E1 -2973.605,E2 -2973.605} C_VEL
LIN {X 0,Y 558.787,Z 703.386,A -85,B 0,C 180,E1 -2975.051,E2 -2975.051} C_VEL
LIN {X 0,Y 558.85,Z 698.609,A -85,B 0,C 180,E1 -2976.499,E2 -2976.499} C_VEL
LIN {X 0,Y 558.95,Z 692.422,A -85,B 0,C 180,E1 -2977.95,E2 -2977.95} C_VEL
LIN {X 0,Y 559.005,Z 684.646,A -85,B 0,C 180,E1 -2979.407,E2 -2979.407} C_VEL
LIN {X 0,Y 559.217,Z 676.368,A -85,B 0,C 180,E1 -2980.683,E2 -2980.683} C_VEL
LIN {X 0,Y 559.362,Z 666.391,A -85,B 0,C 180,E1 -2981.965,E2 -2981.965} C_VEL
LIN {X 0,Y 559.596,Z 656.187,A -85,B 0,C 180,E1 -2983.065,E2 -2983.065} C_VEL
LIN {X 0,Y 559.862,Z 644.019,A -85,B 0,C 180,E1 -2984.169,E2 -2984.169} C_VEL
LIN {X 0,Y 560.123,Z 631.688,A -85,B 0,C 180,E1 -2985.1,E2 -2985.1} C_VEL
LIN {X 0,Y 560.359,Z 618.51,A -85,B 0,C 180,E1 -2985.924,E2 -2985.924} C_VEL
LIN {X 0,Y 560.677,Z 603.826,A -85,B 0,C 180,E1 -2986.663,E2 -2986.663} C_VEL
LIN {X 0,Y 560.916,Z 589.614,A -85,B 0,C 180,E1 -2987.218,E2 -2987.218} C_VEL
LIN {X 0,Y 561.142,Z 575.248,A -85,B 0,C 180,E1 -2987.635,E2 -2987.635} C_VEL
LIN {X 0,Y 561.227,Z 560.813,A -85,B 0,C 180,E1 -2987.921,E2 -2987.921} C_VEL
LIN {X 0,Y 561.782,Z 406.846,A -85,B 0,C 180,E1 -2989.949,E2 -2989.949} C_VEL
LIN {X 0,Y 560.241,Z 398.88,A -85,B 0,C 180,E1 -2990.113,E2 -2990.113} C_VEL
LIN {X 0,Y 560.648,Z 374.764,A -85,B 0,C 180,E1 -2993.062,E2 -2993.062} C_VEL
LIN {X 0,Y 561.004,Z 354.32,A -85,B 0,C 180,E1 -2995.58,E2 -2995.58} C_VEL
LIN {X 0,Y 560.66,Z 350.91,A -85,B 0,C 180,E1 -2996.023,E2 -2996.023} C_VEL
LIN {X 0,Y 559.121,Z 344.466,A -85,B 0,C 180,E1 -2996.93,E2 -2996.93} C_VEL
LIN {X 0,Y 559.14,Z 344.46,A -85,B 0,C 180,E1 -2999.856,E2 -2999.856} C_VEL
LIN {X 0,Y 559.152,Z 344.46,A -85,B 0,C 180,E1 -3002.716,E2 -3002.716} C_VEL
LIN {X 0,Y 559.115,Z 344.46,A -85,B 0,C 180,E1 -3005.325,E2 -3005.325} C_VEL
LIN {X 0,Y 559.124,Z 344.463,A -85,B 0,C 180,E1 -3008.018,E2 -3008.018} C_VEL
LIN {X 0,Y 559.126,Z 344.46,A -85,B 0,C 180,E1 -3010.815,E2 -3010.815} C_VEL
LIN {X 0,Y 559.129,Z 344.458,A -85,B 0,C 180,E1 -3013.195,E2 -3013.195} C_VEL
LIN {X 0,Y 559.123,Z 344.46,A -85,B 0,C 180,E1 -3015.764,E2 -3015.764} C_VEL
LIN {X 0,Y 559.12,Z 344.466,A -85,B 0,C 180,E1 -3018.226,E2 -3018.226} C_VEL
LIN {X 0,Y 559.169,Z 344.452,A -85,B 0,C 180,E1 -3021.193,E2 -3021.193} C_VEL
LIN {X 0,Y 559.116,Z 344.457,A -85,B 0,C 180,E1 -3023.788,E2 -3023.788} C_VEL
LIN {X 0,Y 559.16,Z 344.462,A -85,B 0,C 180,E1 -3026.425,E2 -3026.425} C_VEL
LIN {X 0,Y 559.149,Z 344.451,A -85,B 0,C 180,E1 -3028.981,E2 -3028.981} C_VEL
LIN {X 0,Y 559.133,Z 344.456,A -85,B 0,C 180,E1 -3031.626,E2 -3031.626} C_VEL
LIN {X 0,Y 559.16,Z 344.455,A -85,B 0,C 180,E1 -3033.902,E2 -3033.902} C_VEL
LIN {X 0,Y 559.135,Z 344.463,A -85,B 0,C 180,E1 -3036.573,E2 -3036.573} C_VEL
LIN {X 0,Y 559.173,Z 344.451,A -85,B 0,C 180,E1 -3039.395,E2 -3039.395} C_VEL
LIN {X 0,Y 559.125,Z 344.458,A -85,B 0,C 180,E1 -3041.685,E2 -3041.685} C_VEL
LIN {X 0,Y 559.139,Z 344.458,A -85,B 0,C 180,E1 -3043.947,E2 -3043.947} C_VEL
LIN {X 0,Y 559.157,Z 344.459,A -85,B 0,C 180,E1 -3046.184,E2 -3046.184} C_VEL
LIN {X 0,Y 559.192,Z 344.45,A -85,B 0,C 180,E1 -3049.134,E2 -3049.134} C_VEL
LIN {X 0,Y 559.191,Z 344.452,A -85,B 0,C 180,E1 -3052.054,E2 -3052.054} C_VEL
LIN {X 0,Y 559.238,Z 344.444,A -85,B 0,C 180,E1 -3054.953,E2 -3054.953} C_VEL
LIN {X 0,Y 559.252,Z 344.443,A -85,B 0,C 180,E1 -3057.84,E2 -3057.84} C_VEL
LIN {X 0,Y 559.268,Z 344.445,A -85,B 0,C 180,E1 -3060.72,E2 -3060.72} C_VEL
LIN {X 0,Y 559.225,Z 344.447,A -85,B 0,C 180,E1 -3062.882,E2 -3062.882} C_VEL
LIN {X 0,Y 559.215,Z 344.447,A -85,B 0,C 180,E1 -3065.771,E2 -3065.771} C_VEL
LIN {X 0,Y 559.168,Z 344.459,A -85,B 0,C 180,E1 -3068.675,E2 -3068.675} C_VEL
LIN {X 0,Y 559.207,Z 344.446,A -85,B 0,C 180,E1 -3071.601,E2 -3071.601} C_VEL
LIN {X 0,Y 559.204,Z 344.456,A -85,B 0,C 180,E1 -3074.596,E2 -3074.596} C_VEL
LIN {X 0,Y 559.14,Z 344.455,A -85,B 0,C 180,E1 -3077.558,E2 -3077.558} C_VEL
LIN {X 0,Y 559.168,Z 344.448,A -85,B 0,C 180,E1 -3079.838,E2 -3079.838} C_VEL
LIN {X 0,Y 559.142,Z 344.459,A -85,B 0,C 180,E1 -3082.153,E2 -3082.153} C_VEL
LIN {X 0,Y 559.144,Z 344.452,A -85,B 0,C 180,E1 -3085.179,E2 -3085.179} C_VEL
LIN {X 0,Y 559.137,Z 344.463,A -85,B 0,C 180,E1 -3088.375,E2 -3088.375} C_VEL
LIN {X 0,Y 559.14,Z 344.456,A -85,B 0,C 180,E1 -3090.615,E2 -3090.615} C_VEL
LIN {X 0,Y 558.479,Z 344.538,A -85,B 0,C 180,E1 -3091.216,E2 -3091.216} C_VEL
LIN {X 0,Y 555.615,Z 344.897,A -85,B 0,C 180,E1 -3092.192,E2 -3092.192} C_VEL
LIN {X 0,Y 553.198,Z 345.199,A -85,B 0,C 180,E1 -3092.978,E2 -3092.978} C_VEL
LIN {X 0,Y 552.171,Z 345.325,A -85,B 0,C 180,E1 -3093.584,E2 -3093.584} C_VEL
LIN {X 0,Y 552.093,Z 345.335,A -85,B 0,C 180,E1 -3093.79,E2 -3093.79} C_VEL
LIN {X 0,Y 552.1,Z 345.34,A -85,B 0,C 180,E1 -3096.748,E2 -3096.748} C_VEL
LIN {X 0,Y 552.13,Z 345.327,A -85,B 0,C 180,E1 -3099.528,E2 -3099.528} C_VEL
LIN {X 0,Y 552.112,Z 345.338,A -85,B 0,C 180,E1 -3102.428,E2 -3102.428} C_VEL
LIN {X 0,Y 552.095,Z 345.333,A -85,B 0,C 180,E1 -3105.562,E2 -3105.562} C_VEL
LIN {X 0,Y 552.112,Z 345.34,A -85,B 0,C 180,E1 -3108.68,E2 -3108.68} C_VEL
LIN {X 0,Y 552.118,Z 345.332,A -85,B 0,C 180,E1 -3111.411,E2 -3111.411} C_VEL
LIN {X 0,Y 552.078,Z 345.341,A -85,B 0,C 180,E1 -3114.156,E2 -3114.156} C_VEL
LIN {X 0,Y 552.142,Z 345.353,A -85,B 0,C 180,E1 -3116.27,E2 -3116.27} C_VEL
LIN {X 0,Y 553.364,Z 352.057,A -85,B 0,C 180,E1 -3117.332,E2 -3117.332} C_VEL
LIN {X 0,Y 553.054,Z 368.068,A -85,B 0,C 180,E1 -3119.675,E2 -3119.675} C_VEL
LIN {X 0,Y 555.15,Z 377.729,A -85,B 0,C 180,E1 -3119.887,E2 -3119.887} C_VEL
LIN {X 0,Y 554.435,Z 533.074,A -85,B 0,C 180,E1 -3121.966,E2 -3121.966} C_VEL
LIN {X 0,Y 554.266,Z 549.008,A -85,B 0,C 180,E1 -3122.337,E2 -3122.337} C_VEL
LIN {X 0,Y 553.989,Z 563.616,A -85,B 0,C 180,E1 -3122.825,E2 -3122.825} C_VEL
LIN {X 0,Y 553.696,Z 577.16,A -85,B 0,C 180,E1 -3123.421,E2 -3123.421} C_VEL
LIN {X 0,Y 553.388,Z 591.871,A -85,B 0,C 180,E1 -3124.237,E2 -3124.237} C_VEL
LIN {X 0,Y 553.054,Z 604.592,A -85,B 0,C 180,E1 -3125.106,E2 -3125.106} C_VEL
LIN {X 0,Y 552.774,Z 617.595,A -85,B 0,C 180,E1 -3126.181,E2 -3126.181} C_VEL
LIN {X 0,Y 552.442,Z 629.493,A -85,B 0,C 180,E1 -3127.367,E2 -3127.367} C_VEL
LIN {X 0,Y 552.208,Z 639.314,A -85,B 0,C 180,E1 -3128.537,E2 -3128.537} C_VEL
LIN {X 0,Y 552.068,Z 648.865,A -85,B 0,C 180,E1 -3129.896,E2 -3129.896} C_VEL
LIN {X 0,Y 551.898,Z 656.684,A -85,B 0,C 180,E1 -3131.244,E2 -3131.244} C_VEL
LIN {X 0,Y 551.815,Z 663.969,A -85,B 0,C 180,E1 -3132.789,E2 -3132.789} C_VEL
LIN {X 0,Y 551.753,Z 668.86,A -85,B 0,C 180,E1 -3134.106,E2 -3134.106} C_VEL
LIN {X 0,Y 551.713,Z 672.889,A -85,B 0,C 180,E1 -3135.497,E2 -3135.497} C_VEL
LIN {X 0,Y 551.664,Z 675.575,A -85,B 0,C 180,E1 -3136.743,E2 -3136.743} C_VEL
LIN {X 0,Y 551.674,Z 677.606,A -85,B 0,C 180,E1 -3138.239,E2 -3138.239} C_VEL
LIN {X 0,Y 551.674,Z 678.438,A -85,B 0,C 180,E1 -3139.726,E2 -3139.726} C_VEL
LIN {X 0,Y 551.668,Z 678.106,A -85,B 0,C 180,E1 -3141.206,E2 -3141.206} C_VEL
LIN {X 0,Y 551.69,Z 676.62,A -85,B 0,C 180,E1 -3142.681,E2 -3142.681} C_VEL
LIN {X 0,Y 551.744,Z 673.963,A -85,B 0,C 180,E1 -3144.151,E2 -3144.151} C_VEL
LIN {X 0,Y 551.75,Z 670.06,A -85,B 0,C 180,E1 -3145.617,E2 -3145.617} C_VEL
LIN {X 0,Y 551.765,Z 664.856,A -85,B 0,C 180,E1 -3147.08,E2 -3147.08} C_VEL
LIN {X 0,Y 551.842,Z 658.254,A -85,B 0,C 180,E1 -3148.54,E2 -3148.54} C_VEL
LIN {X 0,Y 552.006,Z 651.167,A -85,B 0,C 180,E1 -3149.818,E2 -3149.818} C_VEL
LIN {X 0,Y 552.163,Z 642.707,A -85,B 0,C 180,E1 -3151.094,E2 -3151.094} C_VEL
LIN {X 0,Y 552.4,Z 632.586,A -85,B 0,C 180,E1 -3152.37,E2 -3152.37} C_VEL
LIN {X 0,Y 552.651,Z 622.297,A -85,B 0,C 180,E1 -3153.463,E2 -3153.463} C_VEL
LIN {X 0,Y 552.968,Z 610.027,A -85,B 0,C 180,E1 -3154.556,E2 -3154.556} C_VEL
LIN {X 0,Y 553.31,Z 597.778,A -85,B 0,C 180,E1 -3155.467,E2 -3155.467} C_VEL
LIN {X 0,Y 553.593,Z 584.456,A -85,B 0,C 180,E1 -3156.286,E2 -3156.286} C_VEL
LIN {X 0,Y 553.888,Z 569.634,A -85,B 0,C 180,E1 -3157.015,E2 -3157.015} C_VEL
LIN {X 0,Y 554.154,Z 554.526,A -85,B 0,C 180,E1 -3157.584,E2 -3157.584} C_VEL
LIN {X 0,Y 554.428,Z 539.419,A -85,B 0,C 180,E1 -3157.992,E2 -3157.992} C_VEL
LIN {X 0,Y 554.524,Z 524.9,A -85,B 0,C 180,E1 -3158.25,E2 -3158.25} C_VEL
LIN {X 0,Y 555.081,Z 377.431,A -85,B 0,C 180,E1 -3160.21,E2 -3160.21} C_VEL
LIN {X 0,Y 553.096,Z 367.898,A -85,B 0,C 180,E1 -3160.432,E2 -3160.432} C_VEL
LIN {X 0,Y 553.419,Z 352.72,A -85,B 0,C 180,E1 -3162.654,E2 -3162.654} C_VEL
LIN {X 0,Y 552.121,Z 345.339,A -85,B 0,C 180,E1 -3163.855,E2 -3163.855} C_VEL
LIN {X 0,Y 552.113,Z 345.336,A -85,B 0,C 180,E1 -3167.024,E2 -3167.024} C_VEL
LIN {X 0,Y 552.13,Z 345.331,A -85,B 0,C 180,E1 -3170.101,E2 -3170.101} C_VEL
LIN {X 0,Y 552.089,Z 345.335,A -85,B 0,C 180,E1 -3172.451,E2 -3172.451} C_VEL
LIN {X 0,Y 552.09,Z 345.341,A -85,B 0,C 180,E1 -3175.334,E2 -3175.334} C_VEL
LIN {X 0,Y 552.068,Z 345.339,A -85,B 0,C 180,E1 -3178.101,E2 -3178.101} C_VEL
LIN {X 0,Y 552.097,Z 345.333,A -85,B 0,C 180,E1 -3180.61,E2 -3180.61} C_VEL
LIN {X 0,Y 552.118,Z 345.333,A -85,B 0,C 180,E1 -3183.186,E2 -3183.186} C_VEL
LIN {X 0,Y 552.074,Z 345.339,A -85,B 0,C 180,E1 -3185.845,E2 -3185.845} C_VEL
LIN {X 0,Y 552.122,Z 345.333,A -85,B 0,C 180,E1 -3189.06,E2 -3189.06} C_VEL
LIN {X 0,Y 552.08,Z 345.34,A -85,B 0,C 180,E1 -3191.45,E2 -3191.45} C_VEL
LIN {X 0,Y 552.079,Z 345.334,A -85,B 0,C 180,E1 -3194.529,E2 -3194.529} C_VEL
LIN {X 0,Y 552.113,Z 345.339,A -85,B 0,C 180,E1 -3197.587,E2 -3197.587} C_VEL
LIN {X 0,Y 552.13,Z 345.328,A -85,B 0,C 180,E1 -3200.472,E2 -3200.472} C_VEL
LIN {X 0,Y 552.1,Z 345.338,A -85,B 0,C 180,E1 -3203.318,E2 -3203.318} C_VEL
LIN {X 0,Y 552.104,Z 345.335,A -85,B 0,C 180,E1 -3205.937,E2 -3205.937} C_VEL
LIN {X 0,Y 552.124,Z 345.33,A -85,B 0,C 180,E1 -3208.54,E2 -3208.54} C_VEL
LIN {X 0,Y 552.099,Z 345.339,A -85,B 0,C 180,E1 -3211.443,E2 -3211.443} C_VEL
LIN {X 0,Y 552.081,Z 345.327,A -85,B 0,C 180,E1 -3214.353,E2 -3214.353} C_VEL
LIN {X 0,Y 552.097,Z 345.33,A -85,B 0,C 180,E1 -3216.757,E2 -3216.757} C_VEL
LIN {X 0,Y 552.121,Z 345.333,A -85,B 0,C 180,E1 -3219.119,E2 -3219.119} C_VEL
LIN {X 0,Y 552.091,Z 345.341,A -85,B 0,C 180,E1 -3221.443,E2 -3221.443} C_VEL
LIN {X 0,Y 552.105,Z 345.339,A -85,B 0,C 180,E1 -3223.737,E2 -3223.737} C_VEL
LIN {X 0,Y 552.129,Z 345.332,A -85,B 0,C 180,E1 -3226.004,E2 -3226.004} C_VEL
LIN {X 0,Y 552.163,Z 345.323,A -85,B 0,C 180,E1 -3228.993,E2 -3228.993} C_VEL
LIN {X 0,Y 552.116,Z 345.334,A -85,B 0,C 180,E1 -3231.951,E2 -3231.951} C_VEL
LIN {X 0,Y 552.216,Z 345.316,A -85,B 0,C 180,E1 -3234.888,E2 -3234.888} C_VEL
LIN {X 0,Y 552.224,Z 345.323,A -85,B 0,C 180,E1 -3237.812,E2 -3237.812} C_VEL
LIN {X 0,Y 552.228,Z 345.318,A -85,B 0,C 180,E1 -3240,E2 -3240} C_VEL
LIN {X 0,Y 552.191,Z 345.32,A -85,B 0,C 180,E1 -3242.918,E2 -3242.918} C_VEL
LIN {X 0,Y 552.187,Z 345.327,A -85,B 0,C 180,E1 -3245.844,E2 -3245.844} C_VEL
LIN {X 0,Y 552.136,Z 345.327,A -85,B 0,C 180,E1 -3248.786,E2 -3248.786} C_VEL
LIN {X 0,Y 552.159,Z 345.331,A -85,B 0,C 180,E1 -3251.75,E2 -3251.75} C_VEL
LIN {X 0,Y 552.13,Z 345.328,A -85,B 0,C 180,E1 -3254.748,E2 -3254.748} C_VEL
LIN {X 0,Y 552.081,Z 345.34,A -85,B 0,C 180,E1 -3257.789,E2 -3257.789} C_VEL
LIN {X 0,Y 552.125,Z 345.331,A -85,B 0,C 180,E1 -3260.101,E2 -3260.101} C_VEL
LIN {X 0,Y 552.084,Z 345.333,A -85,B 0,C 180,E1 -3262.451,E2 -3262.451} C_VEL
LIN {X 0,Y 552.086,Z 345.339,A -85,B 0,C 180,E1 -3265.334,E2 -3265.334} C_VEL
LIN {X 0,Y 552.064,Z 345.34,A -85,B 0,C 180,E1 -3268.101,E2 -3268.101} C_VEL
LIN {X 0,Y 552.093,Z 345.333,A -85,B 0,C 180,E1 -3270.61,E2 -3270.61} C_VEL
LIN {X 0,Y 552.114,Z 345.333,A -85,B 0,C 180,E1 -3273.186,E2 -3273.186} C_VEL
LIN {X 0,Y 552.07,Z 345.343,A -85,B 0,C 180,E1 -3275.845,E2 -3275.845} C_VEL
LIN {X 0,Y 552.117,Z 345.331,A -85,B 0,C 180,E1 -3279.06,E2 -3279.06} C_VEL
LIN {X 0,Y 552.075,Z 345.342,A -85,B 0,C 180,E1 -3281.45,E2 -3281.45} C_VEL
LIN {X 0,Y 552.074,Z 345.336,A -85,B 0,C 180,E1 -3284.529,E2 -3284.529} C_VEL
LIN {X 0,Y 552.109,Z 345.341,A -85,B 0,C 180,E1 -3287.587,E2 -3287.587} C_VEL
LIN {X 0,Y 552.126,Z 345.331,A -85,B 0,C 180,E1 -3290.472,E2 -3290.472} C_VEL
LIN {X 0,Y 552.095,Z 345.339,A -85,B 0,C 180,E1 -3293.318,E2 -3293.318} C_VEL
LIN {X 0,Y 552.116,Z 345.337,A -85,B 0,C 180,E1 -3295.938,E2 -3295.938} C_VEL
LIN {X 0,Y 552.12,Z 345.331,A -85,B 0,C 180,E1 -3298.54,E2 -3298.54} C_VEL
LIN {X 0,Y 552.095,Z 345.342,A -85,B 0,C 180,E1 -3301.444,E2 -3301.444} C_VEL
LIN {X 0,Y 552.092,Z 345.437,A -85,B 0,C 180,E1 -3302.861,E2 -3302.861} C_VEL
LIN {X 0,Y 554.011,Z 353.541,A -85,B 0,C 180,E1 -3303.991,E2 -3303.991} C_VEL
LIN {X 0,Y 554.068,Z 361.91,A -85,B 0,C 180,E1 -3305.054,E2 -3305.054} C_VEL
LIN {X 0,Y 553.608,Z 385.068,A -85,B 0,C 180,E1 -3307.93,E2 -3307.93} C_VEL
LIN {X 0,Y 553.393,Z 399.106,A -85,B 0,C 180,E1 -3309.631,E2 -3309.631} C_VEL
LIN {X 0,Y 555.159,Z 409.109,A -85,B 0,C 180,E1 -3309.834,E2 -3309.834} C_VEL
LIN {X 0,Y 554.469,Z 565.116,A -85,B 0,C 180,E1 -3311.923,E2 -3311.923} C_VEL
LIN {X 0,Y 554.294,Z 580.698,A -85,B 0,C 180,E1 -3312.284,E2 -3312.284} C_VEL
LIN {X 0,Y 554.008,Z 596.032,A -85,B 0,C 180,E1 -3312.798,E2 -3312.798} C_VEL
LIN {X 0,Y 553.789,Z 609.776,A -85,B 0,C 180,E1 -3313.409,E2 -3313.409} C_VEL
LIN {X 0,Y 553.406,Z 623.249,A -85,B 0,C 180,E1 -3314.155,E2 -3314.155} C_VEL
LIN {X 0,Y 553.078,Z 637.139,A -85,B 0,C 180,E1 -3315.103,E2 -3315.103} C_VEL
LIN {X 0,Y 552.76,Z 649.352,A -85,B 0,C 180,E1 -3316.114,E2 -3316.114} C_VEL
LIN {X 0,Y 552.482,Z 661.508,A -85,B 0,C 180,E1 -3317.324,E2 -3317.324} C_VEL
LIN {X 0,Y 552.215,Z 671.483,A -85,B 0,C 180,E1 -3318.513,E2 -3318.513} C_VEL
LIN {X 0,Y 552.125,Z 680.086,A -85,B 0,C 180,E1 -3319.735,E2 -3319.735} C_VEL
LIN {X 0,Y 551.92,Z 687.742,A -85,B 0,C 180,E1 -3321.026,E2 -3321.026} C_VEL
LIN {X 0,Y 551.837,Z 694.09,A -85,B 0,C 180,E1 -3322.315,E2 -3322.315} C_VEL
LIN {X 0,Y 551.769,Z 699.57,A -85,B 0,C 180,E1 -3323.681,E2 -3323.681} C_VEL
LIN {X 0,Y 551.713,Z 703.386,A -85,B 0,C 180,E1 -3324.884,E2 -3324.884} C_VEL
LIN {X 0,Y 551.731,Z 706.888,A -85,B 0,C 180,E1 -3326.348,E2 -3326.348} C_VEL
LIN {X 0,Y 551.654,Z 709.191,A -85,B 0,C 180,E1 -3327.81,E2 -3327.81} C_VEL
LIN {X 0,Y 551.637,Z 710.348,A -85,B 0,C 180,E1 -3329.27,E2 -3329.27} C_VEL
LIN {X 0,Y 551.637,Z 710.348,A -85,B 0,C 180,E1 -3330.73,E2 -3330.73} C_VEL
LIN {X 0,Y 551.654,Z 709.188,A -85,B 0,C 180,E1 -3332.19,E2 -3332.19} C_VEL
LIN {X 0,Y 551.731,Z 706.885,A -85,B 0,C 180,E1 -3333.652,E2 -3333.652} C_VEL
LIN {X 0,Y 551.713,Z 703.387,A -85,B 0,C 180,E1 -3335.116,E2 -3335.116} C_VEL
LIN {X 0,Y 551.78,Z 698.609,A -85,B 0,C 180,E1 -3336.582,E2 -3336.582} C_VEL
LIN {X 0,Y 551.876,Z 692.421,A -85,B 0,C 180,E1 -3338.053,E2 -3338.053} C_VEL
LIN {X 0,Y 551.95,Z 684.645,A -85,B 0,C 180,E1 -3339.528,E2 -3339.528} C_VEL
LIN {X 0,Y 552.183,Z 676.368,A -85,B 0,C 180,E1 -3340.821,E2 -3340.821} C_VEL
LIN {X 0,Y 552.352,Z 666.391,A -85,B 0,C 180,E1 -3342.119,E2 -3342.119} C_VEL
LIN {X 0,Y 552.608,Z 656.186,A -85,B 0,C 180,E1 -3343.234,E2 -3343.234} C_VEL
LIN {X 0,Y 552.907,Z 644.019,A -85,B 0,C 180,E1 -3344.351,E2 -3344.351} C_VEL
LIN {X 0,Y 553.249,Z 631.442,A -85,B 0,C 180,E1 -3345.31,E2 -3345.31} C_VEL
LIN {X 0,Y 553.512,Z 618.507,A -85,B 0,C 180,E1 -3346.126,E2 -3346.126} C_VEL
LIN {X 0,Y 553.832,Z 603.824,A -85,B 0,C 180,E1 -3346.875,E2 -3346.875} C_VEL
LIN {X 0,Y 554.147,Z 589.613,A -85,B 0,C 180,E1 -3347.435,E2 -3347.435} C_VEL
LIN {X 0,Y 554.391,Z 574.631,A -85,B 0,C 180,E1 -3347.873,E2 -3347.873} C_VEL
LIN {X 0,Y 554.501,Z 560.409,A -85,B 0,C 180,E1 -3348.152,E2 -3348.152} C_VEL
LIN {X 0,Y 555.063,Z 407.479,A -85,B 0,C 180,E1 -3350.192,E2 -3350.192} C_VEL
LIN {X 0,Y 553.35,Z 398.793,A -85,B 0,C 180,E1 -3350.386,E2 -3350.386} C_VEL
LIN {X 0,Y 553.807,Z 374.555,A -85,B 0,C 180,E1 -3353.364,E2 -3353.364} C_VEL
LIN {X 0,Y 554.155,Z 355.183,A -85,B 0,C 180,E1 -3355.783,E2 -3355.783} C_VEL
LIN {X 0,Y 552.745,Z 348.147,A -85,B 0,C 180,E1 -3356.75,E2 -3356.75} C_VEL
LIN {X 0,Y 552.095,Z 345.34,A -85,B 0,C 180,E1 -3357.162,E2 -3357.162} C_VEL
LIN {X 0,Y 552.11,Z 345.338,A -85,B 0,C 180,E1 -3360.05,E2 -3360.05} C_VEL
LIN {X 0,Y 552.11,Z 345.336,A -85,B 0,C 180,E1 -3362.846,E2 -3362.846} C_VEL
LIN {X 0,Y 552.063,Z 345.339,A -85,B 0,C 180,E1 -3365.438,E2 -3365.438} C_VEL
LIN {X 0,Y 552.088,Z 345.338,A -85,B 0,C 180,E1 -3367.885,E2 -3367.885} C_VEL
LIN {X 0,Y 552.092,Z 345.341,A -85,B 0,C 180,E1 -3370.483,E2 -3370.483} C_VEL
LIN {X 0,Y 552.092,Z 345.334,A -85,B 0,C 180,E1 -3373.482,E2 -3373.482} C_VEL
LIN {X 0,Y 552.071,Z 345.343,A -85,B 0,C 180,E1 -3376.573,E2 -3376.573} C_VEL
LIN {X 0,Y 552.104,Z 345.334,A -85,B 0,C 180,E1 -3379.798,E2 -3379.798} C_VEL
LIN {X 0,Y 552.083,Z 345.343,A -85,B 0,C 180,E1 -3382.336,E2 -3382.336} C_VEL
LIN {X 0,Y 552.076,Z 345.336,A -85,B 0,C 180,E1 -3385.051,E2 -3385.051} C_VEL
LIN {X 0,Y 552.113,Z 345.331,A -85,B 0,C 180,E1 -3387.681,E2 -3387.681} C_VEL
LIN {X 0,Y 552.087,Z 345.336,A -85,B 0,C 180,E1 -3390.234,E2 -3390.234} C_VEL
LIN {X 0,Y 552.094,Z 345.334,A -85,B 0,C 180,E1 -3393.01,E2 -3393.01} C_VEL
LIN {X 0,Y 552.086,Z 345.338,A -85,B 0,C 180,E1 -3395.961,E2 -3395.961} C_VEL
LIN {X 0,Y 552.116,Z 345.331,A -85,B 0,C 180,E1 -3399.12,E2 -3399.12} C_VEL
LIN {X 0,Y 552.085,Z 345.334,A -85,B 0,C 180,E1 -3401.443,E2 -3401.443} C_VEL
LIN {X 0,Y 552.086,Z 345.335,A -85,B 0,C 180,E1 -3403.737,E2 -3403.737} C_VEL
LIN {X 0,Y 552.126,Z 345.333,A -85,B 0,C 180,E1 -3406.004,E2 -3406.004} C_VEL
LIN {X 0,Y 552.161,Z 345.327,A -85,B 0,C 180,E1 -3408.994,E2 -3408.994} C_VEL
LIN {X 0,Y 552.146,Z 345.328,A -85,B 0,C 180,E1 -3411.952,E2 -3411.952} C_VEL
LIN {X 0,Y 552.214,Z 345.32,A -85,B 0,C 180,E1 -3414.889,E2 -3414.889} C_VEL
LIN {X 0,Y 552.223,Z 345.319,A -85,B 0,C 180,E1 -3417.812,E2 -3417.812} C_VEL
LIN {X 0,Y 552.239,Z 345.321,A -85,B 0,C 180,E1 -3420.73,E2 -3420.73} C_VEL
LIN {X 0,Y 552.191,Z 345.322,A -85,B 0,C 180,E1 -3422.919,E2 -3422.919} C_VEL
LIN {X 0,Y 552.186,Z 345.323,A -85,B 0,C 180,E1 -3425.844,E2 -3425.844} C_VEL
LIN {X 0,Y 552.139,Z 345.333,A -85,B 0,C 180,E1 -3428.786,E2 -3428.786} C_VEL
LIN {X 0,Y 552.164,Z 345.324,A -85,B 0,C 180,E1 -3431.751,E2 -3431.751} C_VEL
LIN {X 0,Y 552.139,Z 345.333,A -85,B 0,C 180,E1 -3434.749,E2 -3434.749} C_VEL
LIN {X 0,Y 552.098,Z 345.333,A -85,B 0,C 180,E1 -3437.789,E2 -3437.789} C_VEL
LIN {X 0,Y 552.129,Z 345.327,A -85,B 0,C 180,E1 -3440.102,E2 -3440.102} C_VEL
LIN {X 0,Y 552.093,Z 345.342,A -85,B 0,C 180,E1 -3442.451,E2 -3442.451} C_VEL
LIN {X 0,Y 552.087,Z 345.33,A -85,B 0,C 180,E1 -3445.335,E2 -3445.335} C_VEL
LIN {X 0,Y 552.08,Z 345.338,A -85,B 0,C 180,E1 -3448.1,E2 -3448.1} C_VEL
LIN {X 0,Y 552.104,Z 345.336,A -85,B 0,C 180,E1 -3450.611,E2 -3450.611} C_VEL
LIN {X 0,Y 552.111,Z 345.333,A -85,B 0,C 180,E1 -3453.187,E2 -3453.187} C_VEL
LIN {X 0,Y 552.093,Z 345.335,A -85,B 0,C 180,E1 -3453.79,E2 -3453.79} C_VEL
LIN {X 0,Y 551.443,Z 345.423,A -85,B 0,C 180,E1 -3454.398,E2 -3454.398} C_VEL
LIN {X 0,Y 548.598,Z 345.779,A -85,B 0,C 180,E1 -3455.386,E2 -3455.386} C_VEL
LIN {X 0,Y 546.176,Z 346.08,A -85,B 0,C 180,E1 -3456.182,E2 -3456.182} C_VEL
LIN {X 0,Y 545.127,Z 346.207,A -85,B 0,C 180,E1 -3456.796,E2 -3456.796} C_VEL
LIN {X 0,Y 545.037,Z 346.216,A -85,B 0,C 180,E1 -3457.004,E2 -3457.004} C_VEL
LIN {X 0,Y 545.062,Z 346.211,A -85,B 0,C 180,E1 -3460.144,E2 -3460.144} C_VEL
LIN {X 0,Y 545.027,Z 346.217,A -85,B 0,C 180,E1 -3463.112,E2 -3463.112} C_VEL
LIN {X 0,Y 545.053,Z 346.215,A -85,B 0,C 180,E1 -3466.227,E2 -3466.227} C_VEL
LIN {X 0,Y 545.076,Z 346.214,A -85,B 0,C 180,E1 -3468.885,E2 -3468.885} C_VEL
LIN {X 0,Y 545.082,Z 346.214,A -85,B 0,C 180,E1 -3470.818,E2 -3470.818} C_VEL
LIN {X 0,Y 545.038,Z 346.214,A -85,B 0,C 180,E1 -3473.619,E2 -3473.619} C_VEL
LIN {X 0,Y 545.12,Z 346.279,A -85,B 0,C 180,E1 -3476.054,E2 -3476.054} C_VEL
LIN {X 0,Y 546.375,Z 352.41,A -85,B 0,C 180,E1 -3477.048,E2 -3477.048} C_VEL
LIN {X 0,Y 546.3,Z 364.214,A -85,B 0,C 180,E1 -3478.815,E2 -3478.815} C_VEL
LIN {X 0,Y 546.174,Z 368.224,A -85,B 0,C 180,E1 -3479.405,E2 -3479.405} C_VEL
LIN {X 0,Y 548.489,Z 379.585,A -85,B 0,C 180,E1 -3479.654,E2 -3479.654} C_VEL
LIN {X 0,Y 547.686,Z 532.956,A -85,B 0,C 180,E1 -3481.733,E2 -3481.733} C_VEL
LIN {X 0,Y 547.481,Z 549.243,A -85,B 0,C 180,E1 -3482.117,E2 -3482.117} C_VEL
LIN {X 0,Y 547.181,Z 563.863,A -85,B 0,C 180,E1 -3482.614,E2 -3482.614} C_VEL
LIN {X 0,Y 546.839,Z 578.386,A -85,B 0,C 180,E1 -3483.268,E2 -3483.268} C_VEL
LIN {X 0,Y 546.504,Z 592.499,A -85,B 0,C 180,E1 -3484.072,E2 -3484.072} C_VEL
LIN {X 0,Y 546.125,Z 605.391,A -85,B 0,C 180,E1 -3484.972,E2 -3484.972} C_VEL
LIN {X 0,Y 545.849,Z 616.858,A -85,B 0,C 180,E1 -3485.935,E2 -3485.935} C_VEL
LIN {X 0,Y 545.499,Z 628.193,A -85,B 0,C 180,E1 -3487.062,E2 -3487.062} C_VEL
LIN {X 0,Y 545.226,Z 638.016,A -85,B 0,C 180,E1 -3488.223,E2 -3488.223} C_VEL
LIN {X 0,Y 545.039,Z 646.666,A -85,B 0,C 180,E1 -3489.429,E2 -3489.429} C_VEL
LIN {X 0,Y 544.87,Z 654.894,A -85,B 0,C 180,E1 -3490.797,E2 -3490.797} C_VEL
LIN {X 0,Y 544.778,Z 660.792,A -85,B 0,C 180,E1 -3491.964,E2 -3491.964} C_VEL
LIN {X 0,Y 544.701,Z 667.115,A -85,B 0,C 180,E1 -3493.51,E2 -3493.51} C_VEL
LIN {X 0,Y 544.647,Z 671.905,A -85,B 0,C 180,E1 -3495.044,E2 -3495.044} C_VEL
LIN {X 0,Y 544.566,Z 675.318,A -85,B 0,C 180,E1 -3496.567,E2 -3496.567} C_VEL
LIN {X 0,Y 544.568,Z 677.465,A -85,B 0,C 180,E1 -3498.083,E2 -3498.083} C_VEL
LIN {X 0,Y 544.579,Z 678.409,A -85,B 0,C 180,E1 -3499.591,E2 -3499.591} C_VEL
LIN {X 0,Y 544.561,Z 678.189,A -85,B 0,C 180,E1 -3501.091,E2 -3501.091} C_VEL
LIN {X 0,Y 544.603,Z 676.815,A -85,B 0,C 180,E1 -3502.585,E2 -3502.585} C_VEL
LIN {X 0,Y 544.642,Z 674.24,A -85,B 0,C 180,E1 -3504.075,E2 -3504.075} C_VEL
LIN {X 0,Y 544.641,Z 670.433,A -85,B 0,C 180,E1 -3505.56,E2 -3505.56} C_VEL
LIN {X 0,Y 544.693,Z 665.352,A -85,B 0,C 180,E1 -3507.042,E2 -3507.042} C_VEL
LIN {X 0,Y 544.757,Z 658.884,A -85,B 0,C 180,E1 -3508.522,E2 -3508.522} C_VEL
LIN {X 0,Y 544.949,Z 651.942,A -85,B 0,C 180,E1 -3509.815,E2 -3509.815} C_VEL
LIN {X 0,Y 545.102,Z 643.647,A -85,B 0,C 180,E1 -3511.108,E2 -3511.108} C_VEL
LIN {X 0,Y 545.374,Z 633.712,A -85,B 0,C 180,E1 -3512.4,E2 -3512.4} C_VEL
LIN {X 0,Y 545.655,Z 623.632,A -85,B 0,C 180,E1 -3513.508,E2 -3513.508} C_VEL
LIN {X 0,Y 546.011,Z 611.625,A -85,B 0,C 180,E1 -3514.614,E2 -3514.614} C_VEL
LIN {X 0,Y 546.417,Z 598.337,A -85,B 0,C 180,E1 -3515.628,E2 -3515.628} C_VEL
LIN {X 0,Y 546.732,Z 585.142,A -85,B 0,C 180,E1 -3516.458,E2 -3516.458} C_VEL
LIN {X 0,Y 547.071,Z 570.507,A -85,B 0,C 180,E1 -3517.196,E2 -3517.196} C_VEL
LIN {X 0,Y 547.34,Z 556.395,A -85,B 0,C 180,E1 -3517.748,E2 -3517.748} C_VEL
LIN {X 0,Y 547.658,Z 540.449,A -85,B 0,C 180,E1 -3518.2,E2 -3518.2} C_VEL
LIN {X 0,Y 547.781,Z 526.376,A -85,B 0,C 180,E1 -3518.46,E2 -3518.46} C_VEL
LIN {X 0,Y 548.422,Z 378.572,A -85,B 0,C 180,E1 -3520.452,E2 -3520.452} C_VEL
LIN {X 0,Y 546.248,Z 368.045,A -85,B 0,C 180,E1 -3520.705,E2 -3520.705} C_VEL
LIN {X 0,Y 546.515,Z 353.825,A -85,B 0,C 180,E1 -3522.817,E2 -3522.817} C_VEL
LIN {X 0,Y 545.088,Z 346.214,A -85,B 0,C 180,E1 -3524.061,E2 -3524.061} C_VEL
LIN {X 0,Y 545.059,Z 346.218,A -85,B 0,C 180,E1 -3527.251,E2 -3527.251} C_VEL
LIN {X 0,Y 545.096,Z 346.205,A -85,B 0,C 180,E1 -3530.372,E2 -3530.372} C_VEL
LIN {X 0,Y 545.079,Z 346.216,A -85,B 0,C 180,E1 -3533.56,E2 -3533.56} C_VEL
LIN {X 0,Y 545.06,Z 346.211,A -85,B 0,C 180,E1 -3536.827,E2 -3536.827} C_VEL
LIN {X 0,Y 545.034,Z 346.22,A -85,B 0,C 180,E1 -3539.34,E2 -3539.34} C_VEL
LIN {X 0,Y 545.059,Z 346.212,A -85,B 0,C 180,E1 -3541.915,E2 -3541.915} C_VEL
LIN {X 0,Y 545.055,Z 346.21,A -85,B 0,C 180,E1 -3544.565,E2 -3544.565} C_VEL
LIN {X 0,Y 545.022,Z 346.218,A -85,B 0,C 180,E1 -3547.305,E2 -3547.305} C_VEL
LIN {X 0,Y 545.063,Z 346.208,A -85,B 0,C 180,E1 -3550.143,E2 -3550.143} C_VEL
LIN {X 0,Y 545.021,Z 346.217,A -85,B 0,C 180,E1 -3553.112,E2 -3553.112} C_VEL
LIN {X 0,Y 545.049,Z 346.209,A -85,B 0,C 180,E1 -3556.227,E2 -3556.227} C_VEL
LIN {X 0,Y 545.033,Z 346.214,A -85,B 0,C 180,E1 -3558.88,E2 -3558.88} C_VEL
LIN {X 0,Y 545.049,Z 346.217,A -85,B 0,C 180,E1 -3561.762,E2 -3561.762} C_VEL
LIN {X 0,Y 545.028,Z 346.213,A -85,B 0,C 180,E1 -3564.53,E2 -3564.53} C_VEL
LIN {X 0,Y 545.069,Z 346.212,A -85,B 0,C 180,E1 -3567.211,E2 -3567.211} C_VEL
LIN {X 0,Y 545.066,Z 346.213,A -85,B 0,C 180,E1 -3569.81,E2 -3569.81} C_VEL
LIN {X 0,Y 545.045,Z 346.205,A -85,B 0,C 180,E1 -3572.341,E2 -3572.341} C_VEL
LIN {X 0,Y 545.044,Z 346.203,A -85,B 0,C 180,E1 -3574.816,E2 -3574.816} C_VEL
LIN {X 0,Y 545.038,Z 346.214,A -85,B 0,C 180,E1 -3577.242,E2 -3577.242} C_VEL
LIN {X 0,Y 545.12,Z 346.202,A -85,B 0,C 180,E1 -3580.414,E2 -3580.414} C_VEL
LIN {X 0,Y 545.057,Z 346.215,A -85,B 0,C 180,E1 -3583.52,E2 -3583.52} C_VEL
LIN {X 0,Y 545.085,Z 346.212,A -85,B 0,C 180,E1 -3585.819,E2 -3585.819} C_VEL
LIN {X 0,Y 545.12,Z 346.199,A -85,B 0,C 180,E1 -3588.849,E2 -3588.849} C_VEL
LIN {X 0,Y 545.073,Z 346.213,A -85,B 0,C 180,E1 -3591.846,E2 -3591.846} C_VEL
LIN {X 0,Y 545.173,Z 346.192,A -85,B 0,C 180,E1 -3594.822,E2 -3594.822} C_VEL
LIN {X 0,Y 545.195,Z 346.199,A -85,B 0,C 180,E1 -3597.783,E2 -3597.783} C_VEL
LIN {X 0,Y 545.196,Z 346.194,A -85,B 0,C 180,E1 -3600,E2 -3600} C_VEL
LIN {X 0,Y 545.159,Z 346.196,A -85,B 0,C 180,E1 -3602.956,E2 -3602.956} C_VEL
LIN {X 0,Y 545.137,Z 346.204,A -85,B 0,C 180,E1 -3605.92,E2 -3605.92} C_VEL
LIN {X 0,Y 545.097,Z 346.204,A -85,B 0,C 180,E1 -3608.9,E2 -3608.9} C_VEL
LIN {X 0,Y 545.102,Z 346.207,A -85,B 0,C 180,E1 -3611.905,E2 -3611.905} C_VEL
LIN {X 0,Y 545.082,Z 346.207,A -85,B 0,C 180,E1 -3614.943,E2 -3614.943} C_VEL
LIN {X 0,Y 545.05,Z 346.212,A -85,B 0,C 180,E1 -3618.026,E2 -3618.026} C_VEL
LIN {X 0,Y 545.091,Z 346.205,A -85,B 0,C 180,E1 -3620.372,E2 -3620.372} C_VEL
LIN {X 0,Y 545.075,Z 346.215,A -85,B 0,C 180,E1 -3623.559,E2 -3623.559} C_VEL
LIN {X 0,Y 545.054,Z 346.213,A -85,B 0,C 180,E1 -3626.002,E2 -3626.002} C_VEL
LIN {X 0,Y 545.049,Z 346.211,A -85,B 0,C 180,E1 -3628.74,E2 -3628.74} C_VEL
LIN {X 0,Y 545.059,Z 346.218,A -85,B 0,C 180,E1 -3631.678,E2 -3631.678} C_VEL
LIN {X 0,Y 545.05,Z 346.211,A -85,B 0,C 180,E1 -3634.565,E2 -3634.565} C_VEL
LIN {X 0,Y 545.018,Z 346.219,A -85,B 0,C 180,E1 -3637.305,E2 -3637.305} C_VEL
LIN {X 0,Y 545.059,Z 346.212,A -85,B 0,C 180,E1 -3640.143,E2 -3640.143} C_VEL
LIN {X 0,Y 545.017,Z 346.217,A -85,B 0,C 180,E1 -3643.112,E2 -3643.112} C_VEL
LIN {X 0,Y 545.045,Z 346.214,A -85,B 0,C 180,E1 -3646.226,E2 -3646.226} C_VEL
LIN {X 0,Y 545.029,Z 346.215,A -85,B 0,C 180,E1 -3648.88,E2 -3648.88} C_VEL
LIN {X 0,Y 545.045,Z 346.22,A -85,B 0,C 180,E1 -3651.762,E2 -3651.762} C_VEL
LIN {X 0,Y 545.023,Z 346.215,A -85,B 0,C 180,E1 -3654.53,E2 -3654.53} C_VEL
LIN {X 0,Y 545.065,Z 346.214,A -85,B 0,C 180,E1 -3657.211,E2 -3657.211} C_VEL
LIN {X 0,Y 545.061,Z 346.217,A -85,B 0,C 180,E1 -3659.81,E2 -3659.81} C_VEL
LIN {X 0,Y 545.065,Z 346.339,A -85,B 0,C 180,E1 -3662.626,E2 -3662.626} C_VEL
LIN {X 0,Y 547.301,Z 356.158,A -85,B 0,C 180,E1 -3664.011,E2 -3664.011} C_VEL
LIN {X 0,Y 546.995,Z 374.571,A -85,B 0,C 180,E1 -3666.349,E2 -3666.349} C_VEL
LIN {X 0,Y 546.469,Z 397.842,A -85,B 0,C 180,E1 -3669.249,E2 -3669.249} C_VEL
LIN {X 0,Y 546.444,Z 398.71,A -85,B 0,C 180,E1 -3669.356,E2 -3669.356} C_VEL
LIN {X 0,Y 548.491,Z 409.647,A -85,B 0,C 180,E1 -3669.587,E2 -3669.587} C_VEL
LIN {X 0,Y 547.734,Z 565.523,A -85,B 0,C 180,E1 -3671.701,E2 -3671.701} C_VEL
LIN {X 0,Y 547.525,Z 580.697,A -85,B 0,C 180,E1 -3672.057,E2 -3672.057} C_VEL
LIN {X 0,Y 547.227,Z 596.03,A -85,B 0,C 180,E1 -3672.578,E2 -3672.578} C_VEL
LIN {X 0,Y 546.962,Z 609.779,A -85,B 0,C 180,E1 -3673.195,E2 -3673.195} C_VEL
LIN {X 0,Y 546.53,Z 623.252,A -85,B 0,C 180,E1 -3673.95,E2 -3673.95} C_VEL
LIN {X 0,Y 546.149,Z 637.141,A -85,B 0,C 180,E1 -3674.909,E2 -3674.909} C_VEL
LIN {X 0,Y 545.818,Z 649.353,A -85,B 0,C 180,E1 -3675.934,E2 -3675.934} C_VEL
LIN {X 0,Y 545.511,Z 661.508,A -85,B 0,C 180,E1 -3677.159,E2 -3677.159} C_VEL
LIN {X 0,Y 545.175,Z 672.103,A -85,B 0,C 180,E1 -3678.446,E2 -3678.446} C_VEL
LIN {X 0,Y 545.05,Z 681.295,A -85,B 0,C 180,E1 -3679.788,E2 -3679.788} C_VEL
LIN {X 0,Y 544.845,Z 688.749,A -85,B 0,C 180,E1 -3681.095,E2 -3681.095} C_VEL
LIN {X 0,Y 544.745,Z 695.7,A -85,B 0,C 180,E1 -3682.587,E2 -3682.587} C_VEL
LIN {X 0,Y 544.709,Z 701.162,A -85,B 0,C 180,E1 -3684.075,E2 -3684.075} C_VEL
LIN {X 0,Y 544.606,Z 705.291,A -85,B 0,C 180,E1 -3685.559,E2 -3685.559} C_VEL
LIN {X 0,Y 544.643,Z 708.185,A -85,B 0,C 180,E1 -3687.041,E2 -3687.041} C_VEL
LIN {X 0,Y 544.543,Z 709.91,A -85,B 0,C 180,E1 -3688.521,E2 -3688.521} C_VEL
LIN {X 0,Y 544.538,Z 710.5,A -85,B 0,C 180,E1 -3690,E2 -3690} C_VEL
LIN {X 0,Y 544.543,Z 709.908,A -85,B 0,C 180,E1 -3691.479,E2 -3691.479} C_VEL
LIN {X 0,Y 544.643,Z 708.182,A -85,B 0,C 180,E1 -3692.959,E2 -3692.959} C_VEL
LIN {X 0,Y 544.606,Z 705.289,A -85,B 0,C 180,E1 -3694.441,E2 -3694.441} C_VEL
LIN {X 0,Y 544.707,Z 701.165,A -85,B 0,C 180,E1 -3695.925,E2 -3695.925} C_VEL
LIN {X 0,Y 544.745,Z 695.701,A -85,B 0,C 180,E1 -3697.413,E2 -3697.413} C_VEL
LIN {X 0,Y 544.845,Z 688.745,A -85,B 0,C 180,E1 -3698.905,E2 -3698.905} C_VEL
LIN {X 0,Y 545.074,Z 680.083,A -85,B 0,C 180,E1 -3700.4,E2 -3700.4} C_VEL
LIN {X 0,Y 545.236,Z 670.706,A -85,B 0,C 180,E1 -3701.735,E2 -3701.735} C_VEL
LIN {X 0,Y 545.511,Z 661.508,A -85,B 0,C 180,E1 -3702.84,E2 -3702.84} C_VEL
LIN {X 0,Y 545.827,Z 649.359,A -85,B 0,C 180,E1 -3704.066,E2 -3704.066} C_VEL
LIN {X 0,Y 546.192,Z 636.806,A -85,B 0,C 180,E1 -3705.115,E2 -3705.115} C_VEL
LIN {X 0,Y 546.529,Z 623.251,A -85,B 0,C 180,E1 -3706.05,E2 -3706.05} C_VEL
LIN {X 0,Y 546.951,Z 609.773,A -85,B 0,C 180,E1 -3706.805,E2 -3706.805} C_VEL
LIN {X 0,Y 547.233,Z 596.042,A -85,B 0,C 180,E1 -3707.421,E2 -3707.421} C_VEL
LIN {X 0,Y 547.524,Z 580.717,A -85,B 0,C 180,E1 -3707.943,E2 -3707.943} C_VEL
LIN {X 0,Y 547.726,Z 564.927,A -85,B 0,C 180,E1 -3708.311,E2 -3708.311} C_VEL
LIN {X 0,Y 548.491,Z 409.621,A -85,B 0,C 180,E1 -3710.413,E2 -3710.413} C_VEL
LIN {X 0,Y 546.457,Z 398.613,A -85,B 0,C 180,E1 -3710.655,E2 -3710.655} C_VEL
LIN {X 0,Y 546.986,Z 374.496,A -85,B 0,C 180,E1 -3713.654,E2 -3713.654} C_VEL
LIN {X 0,Y 547.337,Z 356.871,A -85,B 0,C 180,E1 -3715.885,E2 -3715.885} C_VEL
LIN {X 0,Y 545.065,Z 346.277,A -85,B 0,C 180,E1 -3717.375,E2 -3717.375} C_VEL
LIN {X 0,Y 545.056,Z 346.219,A -85,B 0,C 180,E1 -3720.242,E2 -3720.242} C_VEL
LIN {X 0,Y 545.073,Z 346.211,A -85,B 0,C 180,E1 -3723.061,E2 -3723.061} C_VEL
LIN {X 0,Y 545.019,Z 346.217,A -85,B 0,C 180,E1 -3725.671,E2 -3725.671} C_VEL
LIN {X 0,Y 545.045,Z 346.22,A -85,B 0,C 180,E1 -3728.238,E2 -3728.238} C_VEL
LIN {X 0,Y 545.029,Z 346.213,A -85,B 0,C 180,E1 -3731.12,E2 -3731.12} C_VEL
LIN {X 0,Y 545.038,Z 346.219,A -85,B 0,C 180,E1 -3734.131,E2 -3734.131} C_VEL
LIN {X 0,Y 545.017,Z 346.218,A -85,B 0,C 180,E1 -3736.888,E2 -3736.888} C_VEL
LIN {X 0,Y 545.058,Z 346.213,A -85,B 0,C 180,E1 -3739.857,E2 -3739.857} C_VEL
LIN {X 0,Y 545.026,Z 346.215,A -85,B 0,C 180,E1 -3742.695,E2 -3742.695} C_VEL
LIN {X 0,Y 545.072,Z 346.208,A -85,B 0,C 180,E1 -3745.609,E2 -3745.609} C_VEL
LIN {X 0,Y 545.058,Z 346.214,A -85,B 0,C 180,E1 -3748.322,E2 -3748.322} C_VEL
LIN {X 0,Y 545.064,Z 346.209,A -85,B 0,C 180,E1 -3751.257,E2 -3751.257} C_VEL
LIN {X 0,Y 545.055,Z 346.213,A -85,B 0,C 180,E1 -3753.998,E2 -3753.998} C_VEL
LIN {X 0,Y 545.074,Z 346.215,A -85,B 0,C 180,E1 -3756.441,E2 -3756.441} C_VEL
LIN {X 0,Y 545.091,Z 346.206,A -85,B 0,C 180,E1 -3759.628,E2 -3759.628} C_VEL
LIN {X 0,Y 545.054,Z 346.214,A -85,B 0,C 180,E1 -3762.749,E2 -3762.749} C_VEL
LIN {X 0,Y 545.082,Z 346.208,A -85,B 0,C 180,E1 -3765.82,E2 -3765.82} C_VEL
LIN {X 0,Y 545.118,Z 346.206,A -85,B 0,C 180,E1 -3768.85,E2 -3768.85} C_VEL
LIN {X 0,Y 545.095,Z 346.205,A -85,B 0,C 180,E1 -3771.847,E2 -3771.847} C_VEL
LIN {X 0,Y 545.191,Z 346.195,A -85,B 0,C 180,E1 -3774.823,E2 -3774.823} C_VEL
LIN {X 0,Y 545.195,Z 346.194,A -85,B 0,C 180,E1 -3777.784,E2 -3777.784} C_VEL
LIN {X 0,Y 545.209,Z 346.197,A -85,B 0,C 180,E1 -3780.739,E2 -3780.739} C_VEL
LIN {X 0,Y 545.157,Z 346.198,A -85,B 0,C 180,E1 -3782.956,E2 -3782.956} C_VEL
LIN {X 0,Y 545.136,Z 346.202,A -85,B 0,C 180,E1 -3785.92,E2 -3785.92} C_VEL
LIN {X 0,Y 545.1,Z 346.208,A -85,B 0,C 180,E1 -3788.901,E2 -3788.901} C_VEL
LIN {X 0,Y 545.107,Z 346.204,A -85,B 0,C 180,E1 -3791.905,E2 -3791.905} C_VEL
LIN {X 0,Y 545.088,Z 346.209,A -85,B 0,C 180,E1 -3794.944,E2 -3794.944} C_VEL
LIN {X 0,Y 545.064,Z 346.211,A -85,B 0,C 180,E1 -3798.027,E2 -3798.027} C_VEL
LIN {X 0,Y 545.095,Z 346.206,A -85,B 0,C 180,E1 -3800.373,E2 -3800.373} C_VEL
LIN {X 0,Y 545.08,Z 346.207,A -85,B 0,C 180,E1 -3803.56,E2 -3803.56} C_VEL
LIN {X 0,Y 545.044,Z 346.209,A -85,B 0,C 180,E1 -3806.003,E2 -3806.003} C_VEL
LIN {X 0,Y 545.072,Z 346.214,A -85,B 0,C 180,E1 -3808.744,E2 -3808.744} C_VEL
LIN {X 0,Y 545.061,Z 346.207,A -85,B 0,C 180,E1 -3811.679,E2 -3811.679} C_VEL
LIN {X 0,Y 545.06,Z 346.215,A -85,B 0,C 180,E1 -3814.565,E2 -3814.565} C_VEL
LIN {X 0,Y 545.037,Z 346.216,A -85,B 0,C 180,E1 -3817.004,E2 -3817.004} C_VEL
LIN {X 0,Y 544.358,Z 346.299,A -85,B 0,C 180,E1 -3817.62,E2 -3817.62} C_VEL
LIN {X 0,Y 541.502,Z 346.658,A -85,B 0,C 180,E1 -3818.621,E2 -3818.621} C_VEL
LIN {X 0,Y 539.099,Z 346.953,A -85,B 0,C 180,E1 -3819.427,E2 -3819.427} C_VEL
LIN {X 0,Y 538.071,Z 347.081,A -85,B 0,C 180,E1 -3820.05,E2 -3820.05} C_VEL
LIN {X 0,Y 537.99,Z 347.091,A -85,B 0,C 180,E1 -3820.26,E2 -3820.26} C_VEL
LIN {X 0,Y 537.984,Z 347.095,A -85,B 0,C 180,E1 -3822.982,E2 -3822.982} C_VEL
LIN {X 0,Y 538.022,Z 347.087,A -85,B 0,C 180,E1 -3825.927,E2 -3825.927} C_VEL
LIN {X 0,Y 538.027,Z 347.089,A -85,B 0,C 180,E1 -3829.256,E2 -3829.256} C_VEL
LIN {X 0,Y 537.992,Z 347.095,A -85,B 0,C 180,E1 -3832.122,E2 -3832.122} C_VEL
LIN {X 0,Y 537.998,Z 347.097,A -85,B 0,C 180,E1 -3834.915,E2 -3834.915} C_VEL
LIN {X 0,Y 538.067,Z 347.201,A -85,B 0,C 180,E1 -3835.83,E2 -3835.83} C_VEL
LIN {X 0,Y 539.576,Z 354.687,A -85,B 0,C 180,E1 -3837.058,E2 -3837.058} C_VEL
LIN {X 0,Y 539.384,Z 368.677,A -85,B 0,C 180,E1 -3839.137,E2 -3839.137} C_VEL
LIN {X 0,Y 541.772,Z 379.463,A -85,B 0,C 180,E1 -3839.384,E2 -3839.384} C_VEL
LIN {X 0,Y 541.016,Z 523.867,A -85,B 0,C 180,E1 -3841.352,E2 -3841.352} C_VEL
LIN {X 0,Y 540.904,Z 539.795,A -85,B 0,C 180,E1 -3841.637,E2 -3841.637} C_VEL
LIN {X 0,Y 540.617,Z 554.425,A -85,B 0,C 180,E1 -3842.043,E2 -3842.043} C_VEL
LIN {X 0,Y 540.319,Z 568.221,A -85,B 0,C 180,E1 -3842.568,E2 -3842.568} C_VEL
LIN {X 0,Y 539.96,Z 581.497,A -85,B 0,C 180,E1 -3843.213,E2 -3843.213} C_VEL
LIN {X 0,Y 539.6,Z 594.392,A -85,B 0,C 180,E1 -3843.987,E2 -3843.987} C_VEL
LIN {X 0,Y 539.161,Z 607.379,A -85,B 0,C 180,E1 -3844.935,E2 -3844.935} C_VEL
LIN {X 0,Y 538.826,Z 619.723,A -85,B 0,C 180,E1 -3846.022,E2 -3846.022} C_VEL
LIN {X 0,Y 538.44,Z 630.506,A -85,B 0,C 180,E1 -3847.15,E2 -3847.15} C_VEL
LIN {X 0,Y 538.133,Z 640.503,A -85,B 0,C 180,E1 -3848.393,E2 -3848.393} C_VEL
LIN {X 0,Y 537.954,Z 649.577,A -85,B 0,C 180,E1 -3849.745,E2 -3849.745} C_VEL
LIN {X 0,Y 537.806,Z 656.258,A -85,B 0,C 180,E1 -3850.932,E2 -3850.932} C_VEL
LIN {X 0,Y 537.674,Z 663.572,A -85,B 0,C 180,E1 -3852.504,E2 -3852.504} C_VEL
LIN {X 0,Y 537.592,Z 669.244,A -85,B 0,C 180,E1 -3854.066,E2 -3854.066} C_VEL
LIN {X 0,Y 537.544,Z 673.456,A -85,B 0,C 180,E1 -3855.616,E2 -3855.616} C_VEL
LIN {X 0,Y 537.479,Z 676.344,A -85,B 0,C 180,E1 -3857.156,E2 -3857.156} C_VEL
LIN {X 0,Y 537.544,Z 677.999,A -85,B 0,C 180,E1 -3858.69,E2 -3858.69} C_VEL
LIN {X 0,Y 537.478,Z 678.471,A -85,B 0,C 180,E1 -3860.213,E2 -3860.213} C_VEL
LIN {X 0,Y 537.504,Z 677.781,A -85,B 0,C 180,E1 -3861.731,E2 -3861.731} C_VEL
LIN {X 0,Y 537.553,Z 675.885,A -85,B 0,C 180,E1 -3863.243,E2 -3863.243} C_VEL
LIN {X 0,Y 537.538,Z 672.804,A -85,B 0,C 180,E1 -3864.749,E2 -3864.749} C_VEL
LIN {X 0,Y 537.623,Z 668.488,A -85,B 0,C 180,E1 -3866.252,E2 -3866.252} C_VEL
LIN {X 0,Y 537.613,Z 662.865,A -85,B 0,C 180,E1 -3867.752,E2 -3867.752} C_VEL
LIN {X 0,Y 537.803,Z 655.771,A -85,B 0,C 180,E1 -3869.251,E2 -3869.251} C_VEL
LIN {X 0,Y 537.968,Z 648.227,A -85,B 0,C 180,E1 -3870.561,E2 -3870.561} C_VEL
LIN {X 0,Y 538.239,Z 639.199,A -85,B 0,C 180,E1 -3871.871,E2 -3871.871} C_VEL
LIN {X 0,Y 538.54,Z 628.369,A -85,B 0,C 180,E1 -3873.179,E2 -3873.179} C_VEL
LIN {X 0,Y 538.918,Z 617.292,A -85,B 0,C 180,E1 -3874.3,E2 -3874.3} C_VEL
LIN {X 0,Y 539.313,Z 605.202,A -85,B 0,C 180,E1 -3875.328,E2 -3875.328} C_VEL
LIN {X 0,Y 539.67,Z 592.011,A -85,B 0,C 180,E1 -3876.262,E2 -3876.262} C_VEL
LIN {X 0,Y 540.084,Z 579.068,A -85,B 0,C 180,E1 -3877.007,E2 -3877.007} C_VEL
LIN {X 0,Y 540.403,Z 564.945,A -85,B 0,C 180,E1 -3877.661,E2 -3877.661} C_VEL
LIN {X 0,Y 540.72,Z 550.381,A -85,B 0,C 180,E1 -3878.173,E2 -3878.173} C_VEL
LIN {X 0,Y 540.926,Z 535.152,A -85,B 0,C 180,E1 -3878.552,E2 -3878.552} C_VEL
LIN {X 0,Y 541.14,Z 506.931,A -85,B 0,C 180,E1 -3878.966,E2 -3878.966} C_VEL
LIN {X 0,Y 541.803,Z 379.736,A -85,B 0,C 180,E1 -3880.699,E2 -3880.699} C_VEL
LIN {X 0,Y 539.374,Z 368.391,A -85,B 0,C 180,E1 -3880.962,E2 -3880.962} C_VEL
LIN {X 0,Y 539.601,Z 354.945,A -85,B 0,C 180,E1 -3882.984,E2 -3882.984} C_VEL
LIN {X 0,Y 538.055,Z 347.089,A -85,B 0,C 180,E1 -3884.273,E2 -3884.273} C_VEL
LIN {X 0,Y 538.018,Z 347.097,A -85,B 0,C 180,E1 -3887.524,E2 -3887.524} C_VEL
LIN {X 0,Y 538.09,Z 347.082,A -85,B 0,C 180,E1 -3889.881,E2 -3889.881} C_VEL
LIN {X 0,Y 538.013,Z 347.092,A -85,B 0,C 180,E1 -3893.072,E2 -3893.072} C_VEL
LIN {X 0,Y 538.001,Z 347.097,A -85,B 0,C 180,E1 -3895.662,E2 -3895.662} C_VEL
LIN {X 0,Y 538,Z 347.092,A -85,B 0,C 180,E1 -3898.052,E2 -3898.052} C_VEL
LIN {X 0,Y 538.012,Z 347.088,A -85,B 0,C 180,E1 -3900.628,E2 -3900.628} C_VEL
LIN {X 0,Y 538.051,Z 347.086,A -85,B 0,C 180,E1 -3903.283,E2 -3903.283} C_VEL
LIN {X 0,Y 537.967,Z 347.094,A -85,B 0,C 180,E1 -3906.007,E2 -3906.007} C_VEL
LIN {X 0,Y 538.013,Z 347.088,A -85,B 0,C 180,E1 -3908.831,E2 -3908.831} C_VEL
LIN {X 0,Y 537.994,Z 347.094,A -85,B 0,C 180,E1 -3911.874,E2 -3911.874} C_VEL
LIN {X 0,Y 537.998,Z 347.089,A -85,B 0,C 180,E1 -3914.863,E2 -3914.863} C_VEL
LIN {X 0,Y 537.991,Z 347.091,A -85,B 0,C 180,E1 -3917.211,E2 -3917.211} C_VEL
LIN {X 0,Y 538.014,Z 347.086,A -85,B 0,C 180,E1 -3920.418,E2 -3920.418} C_VEL
LIN {X 0,Y 537.995,Z 347.092,A -85,B 0,C 180,E1 -3923.064,E2 -3923.064} C_VEL
LIN {X 0,Y 538.004,Z 347.093,A -85,B 0,C 180,E1 -3925.825,E2 -3925.825} C_VEL
LIN {X 0,Y 538.012,Z 347.088,A -85,B 0,C 180,E1 -3928.498,E2 -3928.498} C_VEL
LIN {X 0,Y 538.022,Z 347.087,A -85,B 0,C 180,E1 -3931.097,E2 -3931.097} C_VEL
LIN {X 0,Y 537.986,Z 347.087,A -85,B 0,C 180,E1 -3933.63,E2 -3933.63} C_VEL
LIN {X 0,Y 538.01,Z 347.086,A -85,B 0,C 180,E1 -3936.122,E2 -3936.122} C_VEL
LIN {X 0,Y 538.04,Z 347.09,A -85,B 0,C 180,E1 -3939.348,E2 -3939.348} C_VEL
LIN {X 0,Y 538.04,Z 347.08,A -85,B 0,C 180,E1 -3942.467,E2 -3942.467} C_VEL
LIN {X 0,Y 538.054,Z 347.091,A -85,B 0,C 180,E1 -3945.63,E2 -3945.63} C_VEL
LIN {X 0,Y 538.08,Z 347.075,A -85,B 0,C 180,E1 -3948.701,E2 -3948.701} C_VEL
LIN {X 0,Y 538.044,Z 347.09,A -85,B 0,C 180,E1 -3951.739,E2 -3951.739} C_VEL
LIN {X 0,Y 538.132,Z 347.069,A -85,B 0,C 180,E1 -3954.754,E2 -3954.754} C_VEL
LIN {X 0,Y 538.167,Z 347.075,A -85,B 0,C 180,E1 -3957.754,E2 -3957.754} C_VEL
LIN {X 0,Y 538.165,Z 347.07,A -85,B 0,C 180,E1 -3960,E2 -3960} C_VEL
LIN {X 0,Y 538.127,Z 347.072,A -85,B 0,C 180,E1 -3962.994,E2 -3962.994} C_VEL
LIN {X 0,Y 538.093,Z 347.08,A -85,B 0,C 180,E1 -3965.997,E2 -3965.997} C_VEL
LIN {X 0,Y 538.05,Z 347.083,A -85,B 0,C 180,E1 -3969.018,E2 -3969.018} C_VEL
LIN {X 0,Y 538.061,Z 347.082,A -85,B 0,C 180,E1 -3972.063,E2 -3972.063} C_VEL
LIN {X 0,Y 538.04,Z 347.086,A -85,B 0,C 180,E1 -3975.144,E2 -3975.144} C_VEL
LIN {X 0,Y 538.006,Z 347.087,A -85,B 0,C 180,E1 -3978.271,E2 -3978.271} C_VEL
LIN {X 0,Y 538.037,Z 347.084,A -85,B 0,C 180,E1 -3980.651,E2 -3980.651} C_VEL
LIN {X 0,Y 538.008,Z 347.093,A -85,B 0,C 180,E1 -3983.877,E2 -3983.877} C_VEL
LIN {X 0,Y 538.013,Z 347.087,A -85,B 0,C 180,E1 -3986.368,E2 -3986.368} C_VEL
LIN {X 0,Y 537.992,Z 347.091,A -85,B 0,C 180,E1 -3988.925,E2 -3988.925} C_VEL
LIN {X 0,Y 538.01,Z 347.093,A -85,B 0,C 180,E1 -3991.887,E2 -3991.887} C_VEL
LIN {X 0,Y 538,Z 347.089,A -85,B 0,C 180,E1 -3994.615,E2 -3994.615} C_VEL
LIN {X 0,Y 537.983,Z 347.095,A -85,B 0,C 180,E1 -3997.878,E2 -3997.878} C_VEL
LIN {X 0,Y 538,Z 347.089,A -85,B 0,C 180,E1 -4000.78,E2 -4000.78} C_VEL
LIN {X 0,Y 538.001,Z 347.092,A -85,B 0,C 180,E1 -4004.071,E2 -4004.071} C_VEL
LIN {X 0,Y 537.98,Z 347.094,A -85,B 0,C 180,E1 -4007.018,E2 -4007.018} C_VEL
LIN {X 0,Y 538.002,Z 347.094,A -85,B 0,C 180,E1 -4009.258,E2 -4009.258} C_VEL
LIN {X 0,Y 537.984,Z 347.095,A -85,B 0,C 180,E1 -4012.121,E2 -4012.121} C_VEL
LIN {X 0,Y 537.989,Z 347.092,A -85,B 0,C 180,E1 -4014.915,E2 -4014.915} C_VEL
LIN {X 0,Y 538.016,Z 347.096,A -85,B 0,C 180,E1 -4017.617,E2 -4017.617} C_VEL
LIN {X 0,Y 538.01,Z 347.092,A -85,B 0,C 180,E1 -4020.238,E2 -4020.238} C_VEL
LIN {X 0,Y 538.04,Z 347.246,A -85,B 0,C 180,E1 -4022.384,E2 -4022.384} C_VEL
LIN {X 0,Y 540.513,Z 358.359,A -85,B 0,C 180,E1 -4023.975,E2 -4023.975} C_VEL
LIN {X 0,Y 540.005,Z 380.529,A -85,B 0,C 180,E1 -4026.815,E2 -4026.815} C_VEL
LIN {X 0,Y 539.561,Z 398.489,A -85,B 0,C 180,E1 -4029.08,E2 -4029.08} C_VEL
LIN {X 0,Y 541.839,Z 410.409,A -85,B 0,C 180,E1 -4029.338,E2 -4029.338} C_VEL
LIN {X 0,Y 541.013,Z 564.748,A -85,B 0,C 180,E1 -4031.453,E2 -4031.453} C_VEL
LIN {X 0,Y 540.753,Z 580.56,A -85,B 0,C 180,E1 -4031.825,E2 -4031.825} C_VEL
LIN {X 0,Y 540.448,Z 594.699,A -85,B 0,C 180,E1 -4032.304,E2 -4032.304} C_VEL
LIN {X 0,Y 540.153,Z 607.744,A -85,B 0,C 180,E1 -4032.88,E2 -4032.88} C_VEL
LIN {X 0,Y 539.705,Z 621.669,A -85,B 0,C 180,E1 -4033.644,E2 -4033.644} C_VEL
LIN {X 0,Y 539.361,Z 634.493,A -85,B 0,C 180,E1 -4034.516,E2 -4034.516} C_VEL
LIN {X 0,Y 538.946,Z 647.218,A -85,B 0,C 180,E1 -4035.558,E2 -4035.558} C_VEL
LIN {X 0,Y 538.612,Z 657.964,A -85,B 0,C 180,E1 -4036.608,E2 -4036.608} C_VEL
LIN {X 0,Y 538.306,Z 667.903,A -85,B 0,C 180,E1 -4037.751,E2 -4037.751} C_VEL
LIN {X 0,Y 538.111,Z 677.622,A -85,B 0,C 180,E1 -4039.083,E2 -4039.083} C_VEL
LIN {X 0,Y 537.824,Z 685.725,A -85,B 0,C 180,E1 -4040.409,E2 -4040.409} C_VEL
LIN {X 0,Y 537.734,Z 692.423,A -85,B 0,C 180,E1 -4041.734,E2 -4041.734} C_VEL
LIN {X 0,Y 537.618,Z 698.605,A -85,B 0,C 180,E1 -4043.243,E2 -4043.243} C_VEL
LIN {X 0,Y 537.574,Z 703.386,A -85,B 0,C 180,E1 -4044.749,E2 -4044.749} C_VEL
LIN {X 0,Y 537.562,Z 706.887,A -85,B 0,C 180,E1 -4046.252,E2 -4046.252} C_VEL
LIN {X 0,Y 537.487,Z 709.19,A -85,B 0,C 180,E1 -4047.752,E2 -4047.752} C_VEL
LIN {X 0,Y 537.438,Z 710.348,A -85,B 0,C 180,E1 -4049.251,E2 -4049.251} C_VEL
LIN {X 0,Y 537.438,Z 710.347,A -85,B 0,C 180,E1 -4050.749,E2 -4050.749} C_VEL
LIN {X 0,Y 537.487,Z 709.186,A -85,B 0,C 180,E1 -4052.248,E2 -4052.248} C_VEL
LIN {X 0,Y 537.562,Z 706.884,A -85,B 0,C 180,E1 -4053.748,E2 -4053.748} C_VEL
LIN {X 0,Y 537.574,Z 703.387,A -85,B 0,C 180,E1 -4055.251,E2 -4055.251} C_VEL
LIN {X 0,Y 537.618,Z 698.609,A -85,B 0,C 180,E1 -4056.757,E2 -4056.757} C_VEL
LIN {X 0,Y 537.734,Z 692.42,A -85,B 0,C 180,E1 -4058.266,E2 -4058.266} C_VEL
LIN {X 0,Y 537.859,Z 684.643,A -85,B 0,C 180,E1 -4059.78,E2 -4059.78} C_VEL
LIN {X 0,Y 538.101,Z 676.367,A -85,B 0,C 180,E1 -4061.107,E2 -4061.107} C_VEL
LIN {X 0,Y 538.358,Z 666.391,A -85,B 0,C 180,E1 -4062.439,E2 -4062.439} C_VEL
LIN {X 0,Y 538.662,Z 656.184,A -85,B 0,C 180,E1 -4063.583,E2 -4063.583} C_VEL
LIN {X 0,Y 539.029,Z 644.018,A -85,B 0,C 180,E1 -4064.729,E2 -4064.729} C_VEL
LIN {X 0,Y 539.471,Z 631.823,A -85,B 0,C 180,E1 -4065.682,E2 -4065.682} C_VEL
LIN {X 0,Y 539.833,Z 618.494,A -85,B 0,C 180,E1 -4066.546,E2 -4066.546} C_VEL
LIN {X 0,Y 540.223,Z 603.751,A -85,B 0,C 180,E1 -4067.313,E2 -4067.313} C_VEL
LIN {X 0,Y 540.596,Z 588.183,A -85,B 0,C 180,E1 -4067.936,E2 -4067.936} C_VEL
LIN {X 0,Y 540.876,Z 573.119,A -85,B 0,C 180,E1 -4068.371,E2 -4068.371} C_VEL
LIN {X 0,Y 541.061,Z 558.168,A -85,B 0,C 180,E1 -4068.652,E2 -4068.652} C_VEL
LIN {X 0,Y 541.799,Z 409.787,A -85,B 0,C 180,E1 -4070.672,E2 -4070.672} C_VEL
LIN {X 0,Y 539.553,Z 398.379,A -85,B 0,C 180,E1 -4070.931,E2 -4070.931} C_VEL
LIN {X 0,Y 540.137,Z 374.532,A -85,B 0,C 180,E1 -4073.941,E2 -4073.941} C_VEL
LIN {X 0,Y 540.5,Z 358.329,A -85,B 0,C 180,E1 -4076.022,E2 -4076.022} C_VEL
LIN {X 0,Y 538.013,Z 347.096,A -85,B 0,C 180,E1 -4077.642,E2 -4077.642} C_VEL
LIN {X 0,Y 538.012,Z 347.095,A -85,B 0,C 180,E1 -4080.627,E2 -4080.627} C_VEL
LIN {X 0,Y 538.019,Z 347.089,A -85,B 0,C 180,E1 -4083.279,E2 -4083.279} C_VEL
LIN {X 0,Y 537.986,Z 347.097,A -85,B 0,C 180,E1 -4086.005,E2 -4086.005} C_VEL
LIN {X 0,Y 538.008,Z 347.09,A -85,B 0,C 180,E1 -4088.831,E2 -4088.831} C_VEL
LIN {X 0,Y 537.999,Z 347.091,A -85,B 0,C 180,E1 -4091.875,E2 -4091.875} C_VEL
LIN {X 0,Y 537.993,Z 347.093,A -85,B 0,C 180,E1 -4094.864,E2 -4094.864} C_VEL
LIN {X 0,Y 537.972,Z 347.094,A -85,B 0,C 180,E1 -4097.21,E2 -4097.21} C_VEL
LIN {X 0,Y 538.006,Z 347.096,A -85,B 0,C 180,E1 -4100.202,E2 -4100.202} C_VEL
LIN {X 0,Y 537.991,Z 347.087,A -85,B 0,C 180,E1 -4103.065,E2 -4103.065} C_VEL
LIN {X 0,Y 538.016,Z 347.088,A -85,B 0,C 180,E1 -4105.827,E2 -4105.827} C_VEL
LIN {X 0,Y 538.008,Z 347.089,A -85,B 0,C 180,E1 -4108.499,E2 -4108.499} C_VEL
LIN {X 0,Y 538.019,Z 347.087,A -85,B 0,C 180,E1 -4111.098,E2 -4111.098} C_VEL
LIN {X 0,Y 538.014,Z 347.087,A -85,B 0,C 180,E1 -4113.632,E2 -4113.632} C_VEL
LIN {X 0,Y 538.01,Z 347.089,A -85,B 0,C 180,E1 -4116.928,E2 -4116.928} C_VEL
LIN {X 0,Y 538.081,Z 347.084,A -85,B 0,C 180,E1 -4120.148,E2 -4120.148} C_VEL
LIN {X 0,Y 537.988,Z 347.09,A -85,B 0,C 180,E1 -4123.298,E2 -4123.298} C_VEL
LIN {X 0,Y 538.051,Z 347.083,A -85,B 0,C 180,E1 -4125.631,E2 -4125.631} C_VEL
LIN {X 0,Y 538.078,Z 347.085,A -85,B 0,C 180,E1 -4128.702,E2 -4128.702} C_VEL
LIN {X 0,Y 538.059,Z 347.081,A -85,B 0,C 180,E1 -4131.739,E2 -4131.739} C_VEL
LIN {X 0,Y 538.148,Z 347.074,A -85,B 0,C 180,E1 -4134.755,E2 -4134.755} C_VEL
LIN {X 0,Y 538.166,Z 347.069,A -85,B 0,C 180,E1 -4137.755,E2 -4137.755} C_VEL
LIN {X 0,Y 538.18,Z 347.072,A -85,B 0,C 180,E1 -4140.749,E2 -4140.749} C_VEL
LIN {X 0,Y 538.124,Z 347.074,A -85,B 0,C 180,E1 -4142.995,E2 -4142.995} C_VEL
LIN {X 0,Y 538.092,Z 347.081,A -85,B 0,C 180,E1 -4145.998,E2 -4145.998} C_VEL
LIN {X 0,Y 538.052,Z 347.085,A -85,B 0,C 180,E1 -4149.018,E2 -4149.018} C_VEL
LIN {X 0,Y 538.067,Z 347.083,A -85,B 0,C 180,E1 -4152.063,E2 -4152.063} C_VEL
LIN {X 0,Y 538.047,Z 347.084,A -85,B 0,C 180,E1 -4155.144,E2 -4155.144} C_VEL
LIN {X 0,Y 538.017,Z 347.093,A -85,B 0,C 180,E1 -4158.271,E2 -4158.271} C_VEL
LIN {X 0,Y 538.04,Z 347.088,A -85,B 0,C 180,E1 -4160.652,E2 -4160.652} C_VEL
LIN {X 0,Y 538.01,Z 347.089,A -85,B 0,C 180,E1 -4163.878,E2 -4163.878} C_VEL
LIN {X 0,Y 537.987,Z 347.091,A -85,B 0,C 180,E1 -4166.37,E2 -4166.37} C_VEL
LIN {X 0,Y 538.034,Z 347.088,A -85,B 0,C 180,E1 -4168.934,E2 -4168.934} C_VEL
LIN {X 0,Y 538.013,Z 347.086,A -85,B 0,C 180,E1 -4171.887,E2 -4171.887} C_VEL
LIN {X 0,Y 538.009,Z 347.092,A -85,B 0,C 180,E1 -4174.617,E2 -4174.617} C_VEL
LIN {X 0,Y 537.99,Z 347.092,A -85,B 0,C 180,E1 -4177.168,E2 -4177.168} C_VEL
LIN {X 0,Y 538.009,Z 347.087,A -85,B 0,C 180,E1 -4179.799,E2 -4179.799} C_VEL
LIN {X 0,Y 537.99,Z 347.091,A -85,B 0,C 180,E1 -4180.26,E2 -4180.26} C_VEL
LIN {X 0,Y 537.328,Z 347.179,A -85,B 0,C 180,E1 -4180.885,E2 -4180.885} C_VEL
LIN {X 0,Y 534.478,Z 347.533,A -85,B 0,C 180,E1 -4181.9,E2 -4181.9} C_VEL
LIN {X 0,Y 532.064,Z 347.835,A -85,B 0,C 180,E1 -4182.717,E2 -4182.717} C_VEL
LIN {X 0,Y 531.025,Z 347.96,A -85,B 0,C 180,E1 -4183.348,E2 -4183.348} C_VEL
LIN {X 0,Y 530.939,Z 347.97,A -85,B 0,C 180,E1 -4183.562,E2 -4183.562} C_VEL
LIN {X 0,Y 530.948,Z 347.976,A -85,B 0,C 180,E1 -4186.504,E2 -4186.504} C_VEL
LIN {X 0,Y 530.966,Z 347.971,A -85,B 0,C 180,E1 -4188.979,E2 -4188.979} C_VEL
LIN {X 0,Y 530.957,Z 347.968,A -85,B 0,C 180,E1 -4191.529,E2 -4191.529} C_VEL
LIN {X 0,Y 530.954,Z 347.974,A -85,B 0,C 180,E1 -4194.38,E2 -4194.38} C_VEL
LIN {X 0,Y 531.019,Z 348.112,A -85,B 0,C 180,E1 -4195.6,E2 -4195.6} C_VEL
LIN {X 0,Y 532.761,Z 356.76,A -85,B 0,C 180,E1 -4197.033,E2 -4197.033} C_VEL
LIN {X 0,Y 532.505,Z 368.614,A -85,B 0,C 180,E1 -4198.839,E2 -4198.839} C_VEL
LIN {X 0,Y 535.16,Z 380.645,A -85,B 0,C 180,E1 -4199.131,E2 -4199.131} C_VEL
LIN {X 0,Y 534.228,Z 529.795,A -85,B 0,C 180,E1 -4201.196,E2 -4201.196} C_VEL
LIN {X 0,Y 534.021,Z 545.455,A -85,B 0,C 180,E1 -4201.533,E2 -4201.533} C_VEL
LIN {X 0,Y 533.759,Z 559.937,A -85,B 0,C 180,E1 -4201.996,E2 -4201.996} C_VEL
LIN {X 0,Y 533.333,Z 574.956,A -85,B 0,C 180,E1 -4202.641,E2 -4202.641} C_VEL
LIN {X 0,Y 532.923,Z 589.198,A -85,B 0,C 180,E1 -4203.428,E2 -4203.428} C_VEL
LIN {X 0,Y 532.498,Z 601.807,A -85,B 0,C 180,E1 -4204.285,E2 -4204.285} C_VEL
LIN {X 0,Y 532.073,Z 614.273,A -85,B 0,C 180,E1 -4205.309,E2 -4205.309} C_VEL
LIN {X 0,Y 531.669,Z 625.669,A -85,B 0,C 180,E1 -4206.43,E2 -4206.43} C_VEL
LIN {X 0,Y 531.266,Z 636.336,A -85,B 0,C 180,E1 -4207.682,E2 -4207.682} C_VEL
LIN {X 0,Y 530.997,Z 646.138,A -85,B 0,C 180,E1 -4209.062,E2 -4209.062} C_VEL
LIN {X 0,Y 530.756,Z 653.92,A -85,B 0,C 180,E1 -4210.363,E2 -4210.363} C_VEL
LIN {X 0,Y 530.616,Z 661.305,A -85,B 0,C 180,E1 -4211.865,E2 -4211.865} C_VEL
LIN {X 0,Y 530.538,Z 667.511,A -85,B 0,C 180,E1 -4213.453,E2 -4213.453} C_VEL
LIN {X 0,Y 530.499,Z 671.139,A -85,B 0,C 180,E1 -4214.636,E2 -4214.636} C_VEL
LIN {X 0,Y 530.419,Z 674.798,A -85,B 0,C 180,E1 -4216.202,E2 -4216.202} C_VEL
LIN {X 0,Y 530.385,Z 677.178,A -85,B 0,C 180,E1 -4217.76,E2 -4217.76} C_VEL
LIN {X 0,Y 530.414,Z 678.352,A -85,B 0,C 180,E1 -4219.31,E2 -4219.31} C_VEL
LIN {X 0,Y 530.356,Z 678.337,A -85,B 0,C 180,E1 -4220.85,E2 -4220.85} C_VEL
LIN {X 0,Y 530.426,Z 677.123,A -85,B 0,C 180,E1 -4222.386,E2 -4222.386} C_VEL
LIN {X 0,Y 530.455,Z 674.748,A -85,B 0,C 180,E1 -4223.916,E2 -4223.916} C_VEL
LIN {X 0,Y 530.435,Z 671.179,A -85,B 0,C 180,E1 -4225.44,E2 -4225.44} C_VEL
LIN {X 0,Y 530.556,Z 666.342,A -85,B 0,C 180,E1 -4226.963,E2 -4226.963} C_VEL
LIN {X 0,Y 530.587,Z 660.144,A -85,B 0,C 180,E1 -4228.482,E2 -4228.482} C_VEL
LIN {X 0,Y 530.848,Z 652.389,A -85,B 0,C 180,E1 -4230,E2 -4230} C_VEL
LIN {X 0,Y 531.051,Z 644.189,A -85,B 0,C 180,E1 -4231.327,E2 -4231.327} C_VEL
LIN {X 0,Y 531.366,Z 634.424,A -85,B 0,C 180,E1 -4232.653,E2 -4232.653} C_VEL
LIN {X 0,Y 531.712,Z 624.476,A -85,B 0,C 180,E1 -4233.789,E2 -4233.789} C_VEL
LIN {X 0,Y 532.171,Z 612.664,A -85,B 0,C 180,E1 -4234.924,E2 -4234.924} C_VEL
LIN {X 0,Y 532.638,Z 599.644,A -85,B 0,C 180,E1 -4235.964,E2 -4235.964} C_VEL
LIN {X 0,Y 533.051,Z 586.679,A -85,B 0,C 180,E1 -4236.815,E2 -4236.815} C_VEL
LIN {X 0,Y 533.477,Z 572.418,A -85,B 0,C 180,E1 -4237.57,E2 -4237.57} C_VEL
LIN {X 0,Y 533.81,Z 557.495,A -85,B 0,C 180,E1 -4238.184,E2 -4238.184} C_VEL
LIN {X 0,Y 534.176,Z 542.304,A -85,B 0,C 180,E1 -4238.636,E2 -4238.636} C_VEL
LIN {X 0,Y 534.321,Z 528.609,A -85,B 0,C 180,E1 -4238.91,E2 -4238.91} C_VEL
LIN {X 0,Y 535.174,Z 380.937,A -85,B 0,C 180,E1 -4240.953,E2 -4240.953} C_VEL
LIN {X 0,Y 532.514,Z 368.577,A -85,B 0,C 180,E1 -4241.249,E2 -4241.249} C_VEL
LIN {X 0,Y 532.818,Z 357.32,A -85,B 0,C 180,E1 -4242.958,E2 -4242.958} C_VEL
LIN {X 0,Y 531.021,Z 347.965,A -85,B 0,C 180,E1 -4244.515,E2 -4244.515} C_VEL
LIN {X 0,Y 530.977,Z 347.973,A -85,B 0,C 180,E1 -4247.724,E2 -4247.724} C_VEL
LIN {X 0,Y 531.03,Z 347.959,A -85,B 0,C 180,E1 -4250.127,E2 -4250.127} C_VEL
LIN {X 0,Y 530.947,Z 347.969,A -85,B 0,C 180,E1 -4252.573,E2 -4252.573} C_VEL
LIN {X 0,Y 530.957,Z 347.97,A -85,B 0,C 180,E1 -4255.06,E2 -4255.06} C_VEL
LIN {X 0,Y 530.966,Z 347.974,A -85,B 0,C 180,E1 -4257.598,E2 -4257.598} C_VEL
LIN {X 0,Y 530.966,Z 347.965,A -85,B 0,C 180,E1 -4260.642,E2 -4260.642} C_VEL
LIN {X 0,Y 530.968,Z 347.971,A -85,B 0,C 180,E1 -4263.774,E2 -4263.774} C_VEL
LIN {X 0,Y 530.921,Z 347.969,A -85,B 0,C 180,E1 -4266.561,E2 -4266.561} C_VEL
LIN {X 0,Y 530.986,Z 347.971,A -85,B 0,C 180,E1 -4269.444,E2 -4269.444} C_VEL
LIN {X 0,Y 530.923,Z 347.971,A -85,B 0,C 180,E1 -4272.462,E2 -4272.462} C_VEL
LIN {X 0,Y 530.97,Z 347.97,A -85,B 0,C 180,E1 -4275.451,E2 -4275.451} C_VEL
LIN {X 0,Y 530.967,Z 347.965,A -85,B 0,C 180,E1 -4278.561,E2 -4278.561} C_VEL
LIN {X 0,Y 530.955,Z 347.973,A -85,B 0,C 180,E1 -4281.529,E2 -4281.529} C_VEL
LIN {X 0,Y 530.95,Z 347.967,A -85,B 0,C 180,E1 -4284.379,E2 -4284.379} C_VEL
LIN {X 0,Y 530.971,Z 347.967,A -85,B 0,C 180,E1 -4287.133,E2 -4287.133} C_VEL
LIN {X 0,Y 530.957,Z 347.971,A -85,B 0,C 180,E1 -4289.802,E2 -4289.802} C_VEL
LIN {X 0,Y 530.966,Z 347.957,A -85,B 0,C 180,E1 -4292.478,E2 -4292.478} C_VEL
LIN {X 0,Y 530.953,Z 347.957,A -85,B 0,C 180,E1 -4294.939,E2 -4294.939} C_VEL
LIN {X 0,Y 530.981,Z 347.968,A -85,B 0,C 180,E1 -4297.898,E2 -4297.898} C_VEL
LIN {X 0,Y 530.986,Z 347.962,A -85,B 0,C 180,E1 -4300.677,E2 -4300.677} C_VEL
LIN {X 0,Y 530.967,Z 347.963,A -85,B 0,C 180,E1 -4303.07,E2 -4303.07} C_VEL
LIN {X 0,Y 531.011,Z 347.966,A -85,B 0,C 180,E1 -4305.435,E2 -4305.435} C_VEL
LIN {X 0,Y 531.038,Z 347.951,A -85,B 0,C 180,E1 -4308.549,E2 -4308.549} C_VEL
LIN {X 0,Y 530.995,Z 347.97,A -85,B 0,C 180,E1 -4311.628,E2 -4311.628} C_VEL
LIN {X 0,Y 531.092,Z 347.945,A -85,B 0,C 180,E1 -4314.685,E2 -4314.685} C_VEL
LIN {X 0,Y 531.138,Z 347.951,A -85,B 0,C 180,E1 -4317.725,E2 -4317.725} C_VEL
LIN {X 0,Y 531.134,Z 347.945,A -85,B 0,C 180,E1 -4320,E2 -4320} C_VEL
LIN {X 0,Y 531.095,Z 347.949,A -85,B 0,C 180,E1 -4323.034,E2 -4323.034} C_VEL
LIN {X 0,Y 531.052,Z 347.956,A -85,B 0,C 180,E1 -4326.077,E2 -4326.077} C_VEL
LIN {X 0,Y 531.012,Z 347.96,A -85,B 0,C 180,E1 -4329.138,E2 -4329.138} C_VEL
LIN {X 0,Y 531.052,Z 347.961,A -85,B 0,C 180,E1 -4331.67,E2 -4331.67} C_VEL
LIN {X 0,Y 531.025,Z 347.958,A -85,B 0,C 180,E1 -4334.952,E2 -4334.952} C_VEL
LIN {X 0,Y 530.969,Z 347.963,A -85,B 0,C 180,E1 -4338.522,E2 -4338.522} C_VEL
LIN {X 0,Y 530.999,Z 347.961,A -85,B 0,C 180,E1 -4340.938,E2 -4340.938} C_VEL
LIN {X 0,Y 530.952,Z 347.968,A -85,B 0,C 180,E1 -4344.226,E2 -4344.226} C_VEL
LIN {X 0,Y 530.968,Z 347.964,A -85,B 0,C 180,E1 -4346.745,E2 -4346.745} C_VEL
LIN {X 0,Y 530.962,Z 347.971,A -85,B 0,C 180,E1 -4349.324,E2 -4349.324} C_VEL
LIN {X 0,Y 530.965,Z 347.968,A -85,B 0,C 180,E1 -4352.1,E2 -4352.1} C_VEL
LIN {X 0,Y 530.96,Z 347.967,A -85,B 0,C 180,E1 -4354.849,E2 -4354.849} C_VEL
LIN {X 0,Y 530.933,Z 347.977,A -85,B 0,C 180,E1 -4357.51,E2 -4357.51} C_VEL
LIN {X 0,Y 530.948,Z 347.967,A -85,B 0,C 180,E1 -4360.436,E2 -4360.436} C_VEL
LIN {X 0,Y 530.926,Z 347.977,A -85,B 0,C 180,E1 -4363.498,E2 -4363.498} C_VEL
LIN {X 0,Y 530.937,Z 347.97,A -85,B 0,C 180,E1 -4366.502,E2 -4366.502} C_VEL
LIN {X 0,Y 530.948,Z 347.976,A -85,B 0,C 180,E1 -4369.564,E2 -4369.564} C_VEL
LIN {X 0,Y 530.938,Z 347.97,A -85,B 0,C 180,E1 -4372.581,E2 -4372.581} C_VEL
LIN {X 0,Y 530.975,Z 347.97,A -85,B 0,C 180,E1 -4375.309,E2 -4375.309} C_VEL
LIN {X 0,Y 530.966,Z 347.971,A -85,B 0,C 180,E1 -4378.032,E2 -4378.032} C_VEL
LIN {X 0,Y 530.988,Z 347.966,A -85,B 0,C 180,E1 -4380.874,E2 -4380.874} C_VEL
LIN {X 0,Y 530.99,Z 348.054,A -85,B 0,C 180,E1 -4382.122,E2 -4382.122} C_VEL
LIN {X 0,Y 533.648,Z 359.526,A -85,B 0,C 180,E1 -4383.796,E2 -4383.796} C_VEL
LIN {X 0,Y 533.277,Z 377.139,A -85,B 0,C 180,E1 -4386.093,E2 -4386.093} C_VEL
LIN {X 0,Y 532.664,Z 398.268,A -85,B 0,C 180,E1 -4388.796,E2 -4388.796} C_VEL
LIN {X 0,Y 535.196,Z 411.268,A -85,B 0,C 180,E1 -4389.085,E2 -4389.085} C_VEL
LIN {X 0,Y 534.298,Z 564.471,A -85,B 0,C 180,E1 -4391.211,E2 -4391.211} C_VEL
LIN {X 0,Y 533.983,Z 580.318,A -85,B 0,C 180,E1 -4391.586,E2 -4391.586} C_VEL
LIN {X 0,Y 533.66,Z 594.462,A -85,B 0,C 180,E1 -4392.071,E2 -4392.071} C_VEL
LIN {X 0,Y 533.314,Z 607.511,A -85,B 0,C 180,E1 -4392.653,E2 -4392.653} C_VEL
LIN {X 0,Y 532.852,Z 621.445,A -85,B 0,C 180,E1 -4393.428,E2 -4393.428} C_VEL
LIN {X 0,Y 532.479,Z 634.219,A -85,B 0,C 180,E1 -4394.302,E2 -4394.302} C_VEL
LIN {X 0,Y 532.004,Z 647.124,A -85,B 0,C 180,E1 -4395.366,E2 -4395.366} C_VEL
LIN {X 0,Y 531.648,Z 657.937,A -85,B 0,C 180,E1 -4396.429,E2 -4396.429} C_VEL
LIN {X 0,Y 531.313,Z 667.902,A -85,B 0,C 180,E1 -4397.587,E2 -4397.587} C_VEL
LIN {X 0,Y 531.081,Z 677.621,A -85,B 0,C 180,E1 -4398.937,E2 -4398.937} C_VEL
LIN {X 0,Y 530.779,Z 685.726,A -85,B 0,C 180,E1 -4400.281,E2 -4400.281} C_VEL
LIN {X 0,Y 530.665,Z 692.422,A -85,B 0,C 180,E1 -4401.623,E2 -4401.623} C_VEL
LIN {X 0,Y 530.549,Z 698.605,A -85,B 0,C 180,E1 -4403.153,E2 -4403.153} C_VEL
LIN {X 0,Y 530.509,Z 703.386,A -85,B 0,C 180,E1 -4404.679,E2 -4404.679} C_VEL
LIN {X 0,Y 530.481,Z 706.887,A -85,B 0,C 180,E1 -4406.202,E2 -4406.202} C_VEL
LIN {X 0,Y 530.408,Z 709.189,A -85,B 0,C 180,E1 -4407.722,E2 -4407.722} C_VEL
LIN {X 0,Y 530.34,Z 710.347,A -85,B 0,C 180,E1 -4409.241,E2 -4409.241} C_VEL
LIN {X 0,Y 530.34,Z 710.347,A -85,B 0,C 180,E1 -4410.759,E2 -4410.759} C_VEL
LIN {X 0,Y 530.408,Z 709.186,A -85,B 0,C 180,E1 -4412.278,E2 -4412.278} C_VEL
LIN {X 0,Y 530.481,Z 706.883,A -85,B 0,C 180,E1 -4413.798,E2 -4413.798} C_VEL
LIN {X 0,Y 530.508,Z 703.386,A -85,B 0,C 180,E1 -4415.321,E2 -4415.321} C_VEL
LIN {X 0,Y 530.549,Z 698.609,A -85,B 0,C 180,E1 -4416.847,E2 -4416.847} C_VEL
LIN {X 0,Y 530.665,Z 692.42,A -85,B 0,C 180,E1 -4418.377,E2 -4418.377} C_VEL
LIN {X 0,Y 530.809,Z 684.642,A -85,B 0,C 180,E1 -4419.911,E2 -4419.911} C_VEL
LIN {X 0,Y 531.056,Z 676.366,A -85,B 0,C 180,E1 -4421.256,E2 -4421.256} C_VEL
LIN {X 0,Y 531.382,Z 666.391,A -85,B 0,C 180,E1 -4422.605,E2 -4422.605} C_VEL
LIN {X 0,Y 531.71,Z 656.144,A -85,B 0,C 180,E1 -4423.764,E2 -4423.764} C_VEL
LIN {X 0,Y 532.122,Z 643.903,A -85,B 0,C 180,E1 -4424.925,E2 -4424.925} C_VEL
LIN {X 0,Y 532.587,Z 630.402,A -85,B 0,C 180,E1 -4425.981,E2 -4425.981} C_VEL
LIN {X 0,Y 533.054,Z 616.623,A -85,B 0,C 180,E1 -4426.861,E2 -4426.861} C_VEL
LIN {X 0,Y 533.444,Z 602.481,A -85,B 0,C 180,E1 -4427.59,E2 -4427.59} C_VEL
LIN {X 0,Y 533.81,Z 587.933,A -85,B 0,C 180,E1 -4428.172,E2 -4428.172} C_VEL
LIN {X 0,Y 534.122,Z 572.861,A -85,B 0,C 180,E1 -4428.612,E2 -4428.612} C_VEL
LIN {X 0,Y 534.332,Z 557.491,A -85,B 0,C 180,E1 -4428.903,E2 -4428.903} C_VEL
LIN {X 0,Y 535.205,Z 411.263,A -85,B 0,C 180,E1 -4430.914,E2 -4430.914} C_VEL
LIN {X 0,Y 532.663,Z 398.182,A -85,B 0,C 180,E1 -4431.21,E2 -4431.21} C_VEL
LIN {X 0,Y 533.282,Z 375.493,A -85,B 0,C 180,E1 -4434.113,E2 -4434.113} C_VEL
LIN {X 0,Y 533.634,Z 359.484,A -85,B 0,C 180,E1 -4436.201,E2 -4436.201} C_VEL
LIN {X 0,Y 530.987,Z 347.972,A -85,B 0,C 180,E1 -4437.907,E2 -4437.907} C_VEL
LIN {X 0,Y 530.966,Z 347.973,A -85,B 0,C 180,E1 -4440.644,E2 -4440.644} C_VEL
LIN {X 0,Y 530.962,Z 347.969,A -85,B 0,C 180,E1 -4443.5,E2 -4443.5} C_VEL
LIN {X 0,Y 530.933,Z 347.976,A -85,B 0,C 180,E1 -4446.152,E2 -4446.152} C_VEL
LIN {X 0,Y 530.961,Z 347.969,A -85,B 0,C 180,E1 -4448.653,E2 -4448.653} C_VEL
LIN {X 0,Y 530.963,Z 347.965,A -85,B 0,C 180,E1 -4451.439,E2 -4451.439} C_VEL
LIN {X 0,Y 530.965,Z 347.973,A -85,B 0,C 180,E1 -4454.549,E2 -4454.549} C_VEL
LIN {X 0,Y 530.918,Z 347.972,A -85,B 0,C 180,E1 -4457.538,E2 -4457.538} C_VEL
LIN {X 0,Y 530.968,Z 347.973,A -85,B 0,C 180,E1 -4460.555,E2 -4460.555} C_VEL
LIN {X 0,Y 530.935,Z 347.965,A -85,B 0,C 180,E1 -4463.44,E2 -4463.44} C_VEL
LIN {X 0,Y 530.999,Z 347.968,A -85,B 0,C 180,E1 -4466.495,E2 -4466.495} C_VEL
LIN {X 0,Y 530.961,Z 347.958,A -85,B 0,C 180,E1 -4469.358,E2 -4469.358} C_VEL
LIN {X 0,Y 530.965,Z 347.965,A -85,B 0,C 180,E1 -4471.543,E2 -4471.543} C_VEL
LIN {X 0,Y 530.969,Z 347.969,A -85,B 0,C 180,E1 -4474.166,E2 -4474.166} C_VEL
LIN {X 0,Y 530.952,Z 347.972,A -85,B 0,C 180,E1 -4476.603,E2 -4476.603} C_VEL
LIN {X 0,Y 530.998,Z 347.963,A -85,B 0,C 180,E1 -4479.062,E2 -4479.062} C_VEL
LIN {X 0,Y 530.972,Z 347.964,A -85,B 0,C 180,E1 -4481.478,E2 -4481.478} C_VEL
LIN {X 0,Y 530.985,Z 347.969,A -85,B 0,C 180,E1 -4484.65,E2 -4484.65} C_VEL
LIN {X 0,Y 531.024,Z 347.958,A -85,B 0,C 180,E1 -4487.775,E2 -4487.775} C_VEL
LIN {X 0,Y 530.978,Z 347.968,A -85,B 0,C 180,E1 -4490.092,E2 -4490.092} C_VEL
LIN {X 0,Y 531.013,Z 347.966,A -85,B 0,C 180,E1 -4492.395,E2 -4492.395} C_VEL
LIN {X 0,Y 531.106,Z 347.952,A -85,B 0,C 180,E1 -4494.685,E2 -4494.685} C_VEL
LIN {X 0,Y 531.138,Z 347.945,A -85,B 0,C 180,E1 -4497.725,E2 -4497.725} C_VEL
LIN {X 0,Y 531.15,Z 347.948,A -85,B 0,C 180,E1 -4500.758,E2 -4500.758} C_VEL
LIN {X 0,Y 531.09,Z 347.949,A -85,B 0,C 180,E1 -4503.035,E2 -4503.035} C_VEL
LIN {X 0,Y 531.051,Z 347.959,A -85,B 0,C 180,E1 -4506.078,E2 -4506.078} C_VEL
LIN {X 0,Y 531.014,Z 347.961,A -85,B 0,C 180,E1 -4509.139,E2 -4509.139} C_VEL
LIN {X 0,Y 531.052,Z 347.954,A -85,B 0,C 180,E1 -4511.671,E2 -4511.671} C_VEL
LIN {X 0,Y 531.035,Z 347.959,A -85,B 0,C 180,E1 -4514.956,E2 -4514.956} C_VEL
LIN {X 0,Y 530.983,Z 347.963,A -85,B 0,C 180,E1 -4517.724,E2 -4517.724} C_VEL
LIN {X 0,Y 531.028,Z 347.954,A -85,B 0,C 180,E1 -4520.127,E2 -4520.127} C_VEL
LIN {X 0,Y 530.947,Z 347.976,A -85,B 0,C 180,E1 -4522.574,E2 -4522.574} C_VEL
LIN {X 0,Y 530.959,Z 347.962,A -85,B 0,C 180,E1 -4525.06,E2 -4525.06} C_VEL
LIN {X 0,Y 530.965,Z 347.965,A -85,B 0,C 180,E1 -4527.599,E2 -4527.599} C_VEL
LIN {X 0,Y 530.972,Z 347.969,A -85,B 0,C 180,E1 -4530.197,E2 -4530.197} C_VEL
LIN {X 0,Y 530.97,Z 347.97,A -85,B 0,C 180,E1 -4532.867,E2 -4532.867} C_VEL
LIN {X 0,Y 530.951,Z 347.963,A -85,B 0,C 180,E1 -4535.621,E2 -4535.621} C_VEL
LIN {X 0,Y 530.966,Z 347.97,A -85,B 0,C 180,E1 -4538.653,E2 -4538.653} C_VEL
LIN {X 0,Y 530.967,Z 347.966,A -85,B 0,C 180,E1 -4541.439,E2 -4541.439} C_VEL
LIN {X 0,Y 530.939,Z 347.97,A -85,B 0,C 180,E1 -4543.562,E2 -4543.562} C_VEL
LIN {X 0,Y 530.271,Z 348.059,A -85,B 0,C 180,E1 -4544.196,E2 -4544.196} C_VEL
LIN {X 0,Y 527.424,Z 348.416,A -85,B 0,C 180,E1 -4545.225,E2 -4545.225} C_VEL
LIN {X 0,Y 525.019,Z 348.716,A -85,B 0,C 180,E1 -4546.053,E2 -4546.053} C_VEL
LIN {X 0,Y 523.987,Z 348.842,A -85,B 0,C 180,E1 -4546.693,E2 -4546.693} C_VEL
LIN {X 0,Y 523.904,Z 348.849,A -85,B 0,C 180,E1 -4546.909,E2 -4546.909} C_VEL
LIN {X 0,Y 523.938,Z 348.845,A -85,B 0,C 180,E1 -4549.919,E2 -4549.919} C_VEL
LIN {X 0,Y 523.909,Z 348.849,A -85,B 0,C 180,E1 -4552.868,E2 -4552.868} C_VEL
LIN {X 0,Y 523.973,Z 349.036,A -85,B 0,C 180,E1 -4555.363,E2 -4555.363} C_VEL
LIN {X 0,Y 525.915,Z 358.464,A -85,B 0,C 180,E1 -4556.947,E2 -4556.947} C_VEL
LIN {X 0,Y 525.707,Z 369.16,A -85,B 0,C 180,E1 -4558.567,E2 -4558.567} C_VEL
LIN {X 0,Y 528.615,Z 382.09,A -85,B 0,C 180,E1 -4558.877,E2 -4558.877} C_VEL
LIN {X 0,Y 527.543,Z 533.862,A -85,B 0,C 180,E1 -4561.014,E2 -4561.014} C_VEL
LIN {X 0,Y 527.299,Z 549.598,A -85,B 0,C 180,E1 -4561.399,E2 -4561.399} C_VEL
LIN {X 0,Y 526.907,Z 563.941,A -85,B 0,C 180,E1 -4561.901,E2 -4561.901} C_VEL
LIN {X 0,Y 526.448,Z 578.517,A -85,B 0,C 180,E1 -4562.576,E2 -4562.576} C_VEL
LIN {X 0,Y 526.021,Z 593.106,A -85,B 0,C 180,E1 -4563.441,E2 -4563.441} C_VEL
LIN {X 0,Y 525.457,Z 606.814,A -85,B 0,C 180,E1 -4564.447,E2 -4564.447} C_VEL
LIN {X 0,Y 525.026,Z 619.063,A -85,B 0,C 180,E1 -4565.541,E2 -4565.541} C_VEL
LIN {X 0,Y 524.54,Z 630.118,A -85,B 0,C 180,E1 -4566.718,E2 -4566.718} C_VEL
LIN {X 0,Y 524.2,Z 639.844,A -85,B 0,C 180,E1 -4567.951,E2 -4567.951} C_VEL
LIN {X 0,Y 523.903,Z 649.267,A -85,B 0,C 180,E1 -4569.382,E2 -4569.382} C_VEL
LIN {X 0,Y 523.678,Z 656.994,A -85,B 0,C 180,E1 -4570.804,E2 -4570.804} C_VEL
LIN {X 0,Y 523.522,Z 664.01,A -85,B 0,C 180,E1 -4572.392,E2 -4572.392} C_VEL
LIN {X 0,Y 523.416,Z 669.631,A -85,B 0,C 180,E1 -4574.023,E2 -4574.023} C_VEL
LIN {X 0,Y 523.382,Z 672.813,A -85,B 0,C 180,E1 -4575.219,E2 -4575.219} C_VEL
LIN {X 0,Y 523.277,Z 675.939,A -85,B 0,C 180,E1 -4576.802,E2 -4576.802} C_VEL
LIN {X 0,Y 523.32,Z 677.827,A -85,B 0,C 180,E1 -4578.379,E2 -4578.379} C_VEL
LIN {X 0,Y 523.308,Z 678.486,A -85,B 0,C 180,E1 -4579.945,E2 -4579.945} C_VEL
LIN {X 0,Y 523.3,Z 677.958,A -85,B 0,C 180,E1 -4581.505,E2 -4581.505} C_VEL
LIN {X 0,Y 523.37,Z 676.278,A -85,B 0,C 180,E1 -4583.059,E2 -4583.059} C_VEL
LIN {X 0,Y 523.386,Z 673.428,A -85,B 0,C 180,E1 -4584.607,E2 -4584.607} C_VEL
LIN {X 0,Y 523.465,Z 669.358,A -85,B 0,C 180,E1 -4586.151,E2 -4586.151} C_VEL
LIN {X 0,Y 523.445,Z 664.042,A -85,B 0,C 180,E1 -4587.692,E2 -4587.692} C_VEL
LIN {X 0,Y 523.644,Z 657.281,A -85,B 0,C 180,E1 -4589.231,E2 -4589.231} C_VEL
LIN {X 0,Y 523.857,Z 650.026,A -85,B 0,C 180,E1 -4590.577,E2 -4590.577} C_VEL
LIN {X 0,Y 524.156,Z 641.353,A -85,B 0,C 180,E1 -4591.921,E2 -4591.921} C_VEL
LIN {X 0,Y 524.526,Z 630.989,A -85,B 0,C 180,E1 -4593.265,E2 -4593.265} C_VEL
LIN {X 0,Y 524.97,Z 620.371,A -85,B 0,C 180,E1 -4594.415,E2 -4594.415} C_VEL
LIN {X 0,Y 525.453,Z 608.832,A -85,B 0,C 180,E1 -4595.469,E2 -4595.469} C_VEL
LIN {X 0,Y 525.897,Z 596.308,A -85,B 0,C 180,E1 -4596.426,E2 -4596.426} C_VEL
LIN {X 0,Y 526.331,Z 584.264,A -85,B 0,C 180,E1 -4597.191,E2 -4597.191} C_VEL
LIN {X 0,Y 526.777,Z 570.346,A -85,B 0,C 180,E1 -4597.908,E2 -4597.908} C_VEL
LIN {X 0,Y 527.135,Z 555.323,A -85,B 0,C 180,E1 -4598.506,E2 -4598.506} C_VEL
LIN {X 0,Y 527.473,Z 540.337,A -85,B 0,C 180,E1 -4598.935,E2 -4598.935} C_VEL
LIN {X 0,Y 527.657,Z 525.416,A -85,B 0,C 180,E1 -4599.212,E2 -4599.212} C_VEL
LIN {X 0,Y 528.565,Z 382.121,A -85,B 0,C 180,E1 -4601.213,E2 -4601.213} C_VEL
LIN {X 0,Y 525.655,Z 368.765,A -85,B 0,C 180,E1 -4601.545,E2 -4601.545} C_VEL
LIN {X 0,Y 525.917,Z 358.473,A -85,B 0,C 180,E1 -4603.131,E2 -4603.131} C_VEL
LIN {X 0,Y 523.974,Z 348.844,A -85,B 0,C 180,E1 -4604.764,E2 -4604.764} C_VEL
LIN {X 0,Y 523.921,Z 348.849,A -85,B 0,C 180,E1 -4607.971,E2 -4607.971} C_VEL
LIN {X 0,Y 523.963,Z 348.838,A -85,B 0,C 180,E1 -4610.411,E2 -4610.411} C_VEL
LIN {X 0,Y 523.913,Z 348.847,A -85,B 0,C 180,E1 -4612.894,E2 -4612.894} C_VEL
LIN {X 0,Y 523.906,Z 348.852,A -85,B 0,C 180,E1 -4615.421,E2 -4615.421} C_VEL
LIN {X 0,Y 523.915,Z 348.847,A -85,B 0,C 180,E1 -4618.002,E2 -4618.002} C_VEL
LIN {X 0,Y 523.94,Z 348.841,A -85,B 0,C 180,E1 -4620.853,E2 -4620.853} C_VEL
LIN {X 0,Y 523.944,Z 348.847,A -85,B 0,C 180,E1 -4623.731,E2 -4623.731} C_VEL
LIN {X 0,Y 523.873,Z 348.847,A -85,B 0,C 180,E1 -4626.396,E2 -4626.396} C_VEL
LIN {X 0,Y 523.921,Z 348.846,A -85,B 0,C 180,E1 -4629.085,E2 -4629.085} C_VEL
LIN {X 0,Y 523.903,Z 348.847,A -85,B 0,C 180,E1 -4632.124,E2 -4632.124} C_VEL
LIN {X 0,Y 523.94,Z 348.845,A -85,B 0,C 180,E1 -4635.311,E2 -4635.311} C_VEL
LIN {X 0,Y 523.927,Z 348.842,A -85,B 0,C 180,E1 -4638.694,E2 -4638.694} C_VEL
LIN {X 0,Y 523.908,Z 348.849,A -85,B 0,C 180,E1 -4641.897,E2 -4641.897} C_VEL
LIN {X 0,Y 523.921,Z 348.844,A -85,B 0,C 180,E1 -4644.912,E2 -4644.912} C_VEL
LIN {X 0,Y 523.939,Z 348.849,A -85,B 0,C 180,E1 -4647.68,E2 -4647.68} C_VEL
LIN {X 0,Y 523.955,Z 348.837,A -85,B 0,C 180,E1 -4650.677,E2 -4650.677} C_VEL
LIN {X 0,Y 523.903,Z 348.838,A -85,B 0,C 180,E1 -4653.724,E2 -4653.724} C_VEL
LIN {X 0,Y 523.913,Z 348.841,A -85,B 0,C 180,E1 -4656.269,E2 -4656.269} C_VEL
LIN {X 0,Y 523.949,Z 348.84,A -85,B 0,C 180,E1 -4658.766,E2 -4658.766} C_VEL
LIN {X 0,Y 523.941,Z 348.844,A -85,B 0,C 180,E1 -4661.22,E2 -4661.22} C_VEL
LIN {X 0,Y 523.925,Z 348.849,A -85,B 0,C 180,E1 -4663.638,E2 -4663.638} C_VEL
LIN {X 0,Y 523.929,Z 348.844,A -85,B 0,C 180,E1 -4666.027,E2 -4666.027} C_VEL
LIN {X 0,Y 524.017,Z 348.826,A -85,B 0,C 180,E1 -4668.394,E2 -4668.394} C_VEL
LIN {X 0,Y 523.958,Z 348.845,A -85,B 0,C 180,E1 -4671.515,E2 -4671.515} C_VEL
LIN {X 0,Y 524.039,Z 348.824,A -85,B 0,C 180,E1 -4674.613,E2 -4674.613} C_VEL
LIN {X 0,Y 524.109,Z 348.827,A -85,B 0,C 180,E1 -4677.694,E2 -4677.694} C_VEL
LIN {X 0,Y 524.103,Z 348.821,A -85,B 0,C 180,E1 -4680,E2 -4680} C_VEL
LIN {X 0,Y 524.037,Z 348.828,A -85,B 0,C 180,E1 -4683.075,E2 -4683.075} C_VEL
LIN {X 0,Y 524.012,Z 348.832,A -85,B 0,C 180,E1 -4686.159,E2 -4686.159} C_VEL
LIN {X 0,Y 523.982,Z 348.837,A -85,B 0,C 180,E1 -4689.262,E2 -4689.262} C_VEL
LIN {X 0,Y 524.001,Z 348.838,A -85,B 0,C 180,E1 -4691.736,E2 -4691.736} C_VEL
LIN {X 0,Y 523.989,Z 348.835,A -85,B 0,C 180,E1 -4695.049,E2 -4695.049} C_VEL
LIN {X 0,Y 523.916,Z 348.845,A -85,B 0,C 180,E1 -4697.97,E2 -4697.97} C_VEL
LIN {X 0,Y 523.959,Z 348.838,A -85,B 0,C 180,E1 -4700.41,E2 -4700.41} C_VEL
LIN {X 0,Y 523.909,Z 348.843,A -85,B 0,C 180,E1 -4702.893,E2 -4702.893} C_VEL
LIN {X 0,Y 523.906,Z 348.851,A -85,B 0,C 180,E1 -4705.421,E2 -4705.421} C_VEL
LIN {X 0,Y 523.911,Z 348.848,A -85,B 0,C 180,E1 -4708.002,E2 -4708.002} C_VEL
LIN {X 0,Y 523.936,Z 348.841,A -85,B 0,C 180,E1 -4710.853,E2 -4710.853} C_VEL
LIN {X 0,Y 523.951,Z 348.847,A -85,B 0,C 180,E1 -4713.733,E2 -4713.733} C_VEL
LIN {X 0,Y 523.868,Z 348.85,A -85,B 0,C 180,E1 -4716.396,E2 -4716.396} C_VEL
LIN {X 0,Y 523.911,Z 348.844,A -85,B 0,C 180,E1 -4719.085,E2 -4719.085} C_VEL
LIN {X 0,Y 523.899,Z 348.848,A -85,B 0,C 180,E1 -4722.124,E2 -4722.124} C_VEL
LIN {X 0,Y 523.936,Z 348.846,A -85,B 0,C 180,E1 -4725.311,E2 -4725.311} C_VEL
LIN {X 0,Y 523.923,Z 348.844,A -85,B 0,C 180,E1 -4728.694,E2 -4728.694} C_VEL
LIN {X 0,Y 523.903,Z 348.852,A -85,B 0,C 180,E1 -4731.897,E2 -4731.897} C_VEL
LIN {X 0,Y 523.92,Z 348.845,A -85,B 0,C 180,E1 -4734.912,E2 -4734.912} C_VEL
LIN {X 0,Y 523.935,Z 348.85,A -85,B 0,C 180,E1 -4737.68,E2 -4737.68} C_VEL
LIN {X 0,Y 523.952,Z 348.843,A -85,B 0,C 180,E1 -4740.677,E2 -4740.677} C_VEL
LIN {X 0,Y 523.949,Z 348.931,A -85,B 0,C 180,E1 -4741.864,E2 -4741.864} C_VEL
LIN {X 0,Y 526.713,Z 360.715,A -85,B 0,C 180,E1 -4743.611,E2 -4743.611} C_VEL
LIN {X 0,Y 526.793,Z 365.845,A -85,B 0,C 180,E1 -4744.304,E2 -4744.304} C_VEL
LIN {X 0,Y 526.158,Z 386.578,A -85,B 0,C 180,E1 -4747.023,E2 -4747.023} C_VEL
LIN {X 0,Y 525.806,Z 398.196,A -85,B 0,C 180,E1 -4748.51,E2 -4748.51} C_VEL
LIN {X 0,Y 528.587,Z 412.963,A -85,B 0,C 180,E1 -4748.838,E2 -4748.838} C_VEL
LIN {X 0,Y 527.574,Z 564.395,A -85,B 0,C 180,E1 -4750.966,E2 -4750.966} C_VEL
LIN {X 0,Y 527.235,Z 580.077,A -85,B 0,C 180,E1 -4751.342,E2 -4751.342} C_VEL
LIN {X 0,Y 526.894,Z 594.226,A -85,B 0,C 180,E1 -4751.833,E2 -4751.833} C_VEL
LIN {X 0,Y 526.464,Z 607.278,A -85,B 0,C 180,E1 -4752.42,E2 -4752.42} C_VEL
LIN {X 0,Y 526.017,Z 621.217,A -85,B 0,C 180,E1 -4753.206,E2 -4753.206} C_VEL
LIN {X 0,Y 525.544,Z 634.505,A -85,B 0,C 180,E1 -4754.129,E2 -4754.129} C_VEL
LIN {X 0,Y 525.047,Z 646.911,A -85,B 0,C 180,E1 -4755.168,E2 -4755.168} C_VEL
LIN {X 0,Y 524.677,Z 657.713,A -85,B 0,C 180,E1 -4756.246,E2 -4756.246} C_VEL
LIN {X 0,Y 524.314,Z 667.719,A -85,B 0,C 180,E1 -4757.419,E2 -4757.419} C_VEL
LIN {X 0,Y 524.031,Z 677.51,A -85,B 0,C 180,E1 -4758.786,E2 -4758.786} C_VEL
LIN {X 0,Y 523.739,Z 685.678,A -85,B 0,C 180,E1 -4760.149,E2 -4760.149} C_VEL
LIN {X 0,Y 523.612,Z 692.422,A -85,B 0,C 180,E1 -4761.51,E2 -4761.51} C_VEL
LIN {X 0,Y 523.48,Z 698.605,A -85,B 0,C 180,E1 -4763.06,E2 -4763.06} C_VEL
LIN {X 0,Y 523.442,Z 703.385,A -85,B 0,C 180,E1 -4764.607,E2 -4764.607} C_VEL
LIN {X 0,Y 523.402,Z 706.886,A -85,B 0,C 180,E1 -4766.15,E2 -4766.15} C_VEL
LIN {X 0,Y 523.332,Z 709.189,A -85,B 0,C 180,E1 -4767.691,E2 -4767.691} C_VEL
LIN {X 0,Y 523.246,Z 710.347,A -85,B 0,C 180,E1 -4769.23,E2 -4769.23} C_VEL
LIN {X 0,Y 523.246,Z 710.346,A -85,B 0,C 180,E1 -4770.77,E2 -4770.77} C_VEL
LIN {X 0,Y 523.332,Z 709.185,A -85,B 0,C 180,E1 -4772.309,E2 -4772.309} C_VEL
LIN {X 0,Y 523.402,Z 706.882,A -85,B 0,C 180,E1 -4773.85,E2 -4773.85} C_VEL
LIN {X 0,Y 523.441,Z 703.386,A -85,B 0,C 180,E1 -4775.393,E2 -4775.393} C_VEL
LIN {X 0,Y 523.48,Z 698.609,A -85,B 0,C 180,E1 -4776.94,E2 -4776.94} C_VEL
LIN {X 0,Y 523.611,Z 692.419,A -85,B 0,C 180,E1 -4778.49,E2 -4778.49} C_VEL
LIN {X 0,Y 523.776,Z 684.582,A -85,B 0,C 180,E1 -4780.046,E2 -4780.046} C_VEL
LIN {X 0,Y 524.013,Z 676.239,A -85,B 0,C 180,E1 -4781.41,E2 -4781.41} C_VEL
LIN {X 0,Y 524.38,Z 666.189,A -85,B 0,C 180,E1 -4782.776,E2 -4782.776} C_VEL
LIN {X 0,Y 524.725,Z 655.91,A -85,B 0,C 180,E1 -4783.951,E2 -4783.951} C_VEL
LIN {X 0,Y 525.21,Z 643.667,A -85,B 0,C 180,E1 -4785.126,E2 -4785.126} C_VEL
LIN {X 0,Y 525.706,Z 630.042,A -85,B 0,C 180,E1 -4786.205,E2 -4786.205} C_VEL
LIN {X 0,Y 526.221,Z 616.382,A -85,B 0,C 180,E1 -4787.087,E2 -4787.087} C_VEL
LIN {X 0,Y 526.669,Z 602.237,A -85,B 0,C 180,E1 -4787.823,E2 -4787.823} C_VEL
LIN {X 0,Y 527.063,Z 587.683,A -85,B 0,C 180,E1 -4788.412,E2 -4788.412} C_VEL
LIN {X 0,Y 527.384,Z 572.103,A -85,B 0,C 180,E1 -4788.871,E2 -4788.871} C_VEL
LIN {X 0,Y 527.623,Z 556.498,A -85,B 0,C 180,E1 -4789.163,E2 -4789.163} C_VEL
